					{Region "WA MANAGER LASTRA DA PICKPOINT"}
					(* Ciclo lastra PRELIEVO lastra da punto di prelievo classico *)	
					WAMANAGER_CICLO_PRELIEVO_LASTRA_PP_RUN:
						(* Controllo che la pinza si libera *)
						IF PinzaConProdottoInPresa AND PinzaInQuotaFuoriIngombro THEN
							CmdExe.RapidStopRequest := 1;
							TFError(ErrPRESENZA_MATERIALE_SUPINZA_CICLO_PRELPACCO,ErrNULL,ADR(CmdExe),ADR(State),ADR(Error),ADR(ErrorLog));
						ELSE					
							Mission^.State :=  MISSION_STATE_PRELIEVO_LASTRA_PP_RUN;
						END_IF
							 
					WAMANAGER_CICLO_PRELIEVO_LASTRA_PP_END:;
						 
					(* Ciclo lastra deposito su rulliera *)
					WAMANAGER_CICLO_DEPOSITO_LASTRA_PP_RUN:
						(* Se ho presenza logica *)
						IF ProductOnGripper = KPRODUCTLOADED THEN
							(* Se è abilitato il controllo della presenza utilizzando la fotocellula *)
							IF AbilitaControlloPHGripPresence THEN
								(* Se NON vedo la fotocellula *)
								IF NOT PinzaConProdottoInPresa AND PinzaInQuotaFuoriIngombro THEN
									TFError(ErrLOADLOST,ErrNULL,ADR(CmdExe),ADR(State),ADR(Error),ADR(ErrorLog));
									CmdExe.RapidStopRequest := 1;
									CmdExe.PhaseStopRequest := 1;
								END_IF
							END_IF
						END_IF		
							
						(* Controllo la presenza del pallet nella Postazione di deposito *)	
						IF (Mission^.TPick = TPICK_LASTRA AND NOT IN.PX_WorkArea[Mission^.PPlace]) AND NOT SimulazioneSenzaPalletFalde THEN
							CmdExe.PhaseStopRequest := 1;
							TFError(ErrPALLETNOTPRESENT,Mission^.PPlace,ADR(CmdExe),ADR(State),ADR(Error),ADR(ErrorLog));
						(* Se non ho alcun errore procedo con la missione *)
						ELSIF CmdExe.RapidStopRequest = 0 THEN
							Mission^.State := MISSION_STATE_DEPOSITO_LASTRA_PP_RUN;
						END_IF	
						 
					WAMANAGER_CICLO_DEPOSITO_LASTRA_PP_END:
						 ProductOnGripper := KNOPRODUCT;
				
					{endregion}

					{Region "WA MANAGER LASTRA WA PAL"}		
					WAMANAGER_CICLO_PRELIEVO_LASTRA_WA_RUN:
						(* Controllo che la pinza si libera *)
						IF ((PX_GripPresenceFiltrata AND NOT PX_GripPresenceOK AND AbilitaControlloPHGripPresence) (*OR ProductOnGripper <> KNOPRODUCT*)) AND PinzaInQuotaFuoriIngombro THEN
							CmdExe.RapidStopRequest := 1;
							TFError(ErrPRESENZA_MATERIALE_SUPINZA_CICLO_PRELPACCO,ErrNULL,ADR(CmdExe),ADR(State),ADR(Error),ADR(ErrorLog));
						ELSE					
							Mission^.State :=  MISSION_STATE_PRELIEVO_LASTRA_WA_RUN;	
							PX_GripPresenceOK := TRUE;		
						END_IF					
					WAMANAGER_CICLO_PRELIEVO_LASTRA_WA_END:
						PX_GripPresenceOK := FALSE;
						ProductOnGripper := KPRODUCTLOADED;												
						
					WAMANAGER_CICLO_DEPOSITO_LASTRA_WA_RUN:
						(* Se ho presenza logica *)
						IF ProductOnGripper = KPRODUCTLOADED THEN
							(* Se è abilitato il controllo della presenza utilizzando la fotocellula *)
							IF AbilitaControlloPHGripPresence THEN
								(* Se NON vedo la fotocellula *)
								IF NOT PX_GripPresenceFiltrata AND PinzaInQuotaFuoriIngombro THEN
									TFError(ErrLOADLOST,ErrNULL,ADR(CmdExe),ADR(State),ADR(Error),ADR(ErrorLog));
									CmdExe.RapidStopRequest := 1;
									CmdExe.PhaseStopRequest := 1;
								END_IF
							END_IF
						END_IF		
							
						(* Controllo la presenza del pallet nella Postazione di deposito *)	
						IF (Mission^.TPick = TPICK_PACK AND NOT IN.PX_WorkArea[Mission^.PPlace]) AND NOT SimulazioneSenzaPalletFalde THEN
							CmdExe.PhaseStopRequest := 1;
							TFError(ErrPALLETNOTPRESENT,Mission^.PPlace,ADR(CmdExe),ADR(State),ADR(Error),ADR(ErrorLog));
						(* Se non ho alcun errore procedo con la missione *)
						ELSIF CmdExe.RapidStopRequest = 0 THEN
							Mission^.State := MISSION_STATE_DEPOSITO_LASTRA_WA_RUN;
						END_IF	
						
					WAMANAGER_CICLO_DEPOSITO_LASTRA_WA_END:
						ProductOnGripper := KNOPRODUCT;
					{endregion}	
{region "DEPALLETTIZZATORE"}	
					(* Ciclo lastra PRELIEVO lastra depallettizzatore *)	
					WAMANAGER_CICLO_PRELIEVO_LASTRA_DEPAL_RUN:
						(* Controllo che la pinza si libera *)
						IF ((PX_GripPresenceFiltrata AND NOT PX_GripPresenceOK AND AbilitaControlloPHGripPresence) OR ProductOnGripper <> KNOPRODUCT) AND PinzaInQuotaFuoriIngombro THEN
							CmdExe.RapidStopRequest := 1;
							TFError(ErrPRESENZA_MATERIALE_SUPINZA_CICLO_PRELPACCO,ErrNULL,ADR(CmdExe),ADR(State),ADR(Error),ADR(ErrorLog));
						ELSE					
							Mission^.State :=  MISSION_STATE_PRELIEVO_LASTRA_DEPAL_RUN;	
							PX_GripPresenceOK := TRUE;		
						END_IF
							 
					WAMANAGER_CICLO_PRELIEVO_LASTRA_DEPAL_END:;
						 
					(* Ciclo lastra deposito su rulliera *)
					WAMANAGER_CICLO_DEPOSITO_LASTRA_DEPAL_RUN:
						(* Se ho presenza logica *)
						IF ProductOnGripper = KPRODUCTLOADED THEN
							(* Se è abilitato il controllo della presenza utilizzando la fotocellula *)
							IF AbilitaControlloPHGripPresence THEN
								(* Se NON vedo la fotocellula *)
								IF NOT PX_GripPresenceFiltrata AND PinzaInQuotaFuoriIngombro THEN
									TFError(ErrLOADLOST,ErrNULL,ADR(CmdExe),ADR(State),ADR(Error),ADR(ErrorLog));
									CmdExe.RapidStopRequest := 1;
									CmdExe.PhaseStopRequest := 1;
								END_IF
							END_IF
						END_IF		
							
						(* Controllo la presenza del pallet nella Postazione di deposito *)	
						IF (Mission^.TPick = TPICK_PACK AND NOT IN.PX_WorkArea[Mission^.PPlace]) AND NOT SimulazioneSenzaPalletFalde THEN
							CmdExe.PhaseStopRequest := 1;
							TFError(ErrPALLETNOTPRESENT,Mission^.PPlace,ADR(CmdExe),ADR(State),ADR(Error),ADR(ErrorLog));
						(* Se non ho alcun errore procedo con la missione *)
						ELSIF CmdExe.RapidStopRequest = 0 THEN
							Mission^.State := MISSION_STATE_DEPOSITO_LASTRA_DEPAL_RUN;
						END_IF	
						 
					WAMANAGER_CICLO_DEPOSITO_LASTRA_DEPAL_END:
						 ProductOnGripper := KNOPRODUCT;
							  
					(* Ciclo deposito FALDA su magazzino dedicato dopo prelievo misto da postazione *)
					WAMANAGER_CICLO_DEPOSITO_FALDA_DEPAL_RUN:
						 	
						(* Se ho presenza logica *)
						(*IF ProductOnGripper = KPRODUCTLOADED THEN
							(* Se è abilitato il controllo della presenza utilizzando la fotocellula *)
							IF AbilitaControlloPHGripPresence THEN
								(* Se NON vedo la fotocellula *)
								IF NOT PX_GripPresenceFiltrata AND PinzaInQuotaFuoriIngombro THEN
									TFError(ErrLOADLOST,ErrNULL,ADR(CmdExe),ADR(State),ADR(Error),ADR(ErrorLog));
									CmdExe.RapidStopRequest := 1;
									CmdExe.PhaseStopRequest := 1;
								END_IF
							END_IF
						END_IF*)
							
						IF CmdExe.RapidStopRequest = 0 THEN
							Mission^.State := MISSION_STATE_DEPOSITO_FALDA_DEPAL_RUN;
						END_IF		 
														 
					WAMANAGER_CICLO_DEPOSITO_FALDA_DEPAL_END:
						ProductOnGripper := KNOPRODUCT;	
{endregion}													
				END_CASE
				
{region "CASE MISSION"}		
				(* Eseguo il passo della Missione *)
				CASE Mission^.State OF					
					MISSION_STATE_NOP:
						(* Missione di NOP - WorkFlow  *)
						IF MissionStateCase^.Mission <> MISSION_STATE_NOP THEN
							MissionStateCase^.NCase := 0;
							MissionStateCase^.Mission := MISSION_STATE_NOP;
						END_IF
						
						CASE MissionStateCase^.NCase OF
							(* Case 0 - *)
							0:	
								MissionStateCase^.NCase := 0;
						END_CASE
												
					MISSION_STATE_INIT:
						(* Missione di INIT - WorkFlow  *)
						IF MissionStateCase^.Mission <> MISSION_STATE_INIT THEN
							MissionStateCase^.NCase := 0;
							MissionStateCase^.Mission := MISSION_STATE_INIT;
						END_IF
				{Region "MISSION RIPOSO"}						
					MISSION_STATE_VAIaRIPOSO_RUN:// Assegnato al WorkFlow 2
						(* Missione di RIPOSO - WorkFlow  *)
						NumeroWF := 2;//Numero del WorkFlow
						IF ((MissionStateCase^.Mission <> MISSION_STATE_VAIaRIPOSO_RUN AND MissionStateCase^.Mission <> MISSION_STATE_VAIaRIPOSO_END) AND NOT ForzaPrelievoPaccoDuranteCicloDiRiposo)  THEN
							MissionStateCase^.NCase := 0;
							MissionStateCase^.Mission := MISSION_STATE_VAIaRIPOSO_RUN;
						ELSIF ForzaPrelievoPaccoDuranteCicloDiRiposo THEN
							WorkFlow[NumeroWF].Enable := FALSE;
							MissionStateCase^.NCase := 10;
							Ciclo_Di_Riposo.Stato := INTERROTTO;
						END_IF	
												
						CASE MissionStateCase^.NCase OF
							(* Case 0 - Attivazione e inizializzazione del Workflow*)
							0:	WorkFlow[NumeroWF].Enable := TRUE;
								TFWorkFlowCase(ADR(WorkFlow[NumeroWF]),0,WorkflowCase_JMP);
								MissionStateCase^.NCase := 1;
				
							(* Case 1 - Attesa di un eventuale stop rapido/stop in fase o attesa del completamento/errore workflow *)
							1:	IF CmdExe.RapidStopRequest > 0 OR
									(NOT WorkFlow[NumeroWF].Enable OR WorkFlow[NumeroWF].WFCase = StateWF_ERROR) THEN
									MissionStateCase^.NCase := 2;
								END_IF;
				
							(* Case 2 - Wait WF End *)
							2: IF (NOT WorkFlow[NumeroWF].Enable OR WorkFlow[NumeroWF].State = StateWF_END OR WorkFlow[NumeroWF].WFCase = StateWF_ERROR) THEN
									WorkFlow[NumeroWF].Enable := FALSE;
									IF WorkFlow[NumeroWF].WFCase = StateWF_ERROR THEN
										IF Warning.Code <> ErrNULL THEN
											TFError(Warning.Code,ErrNULL,ADR(CmdExe),ADR(State),ADR(Error),ADR(ErrorLog));
										ELSE
											TFError(ErrWF,ErrNULL,ADR(CmdExe),ADR(State),ADR(Error),ADR(ErrorLog));
										END_IF
									ELSIF WorkFlow[NumeroWF].State = StateWF_END THEN
										MissionStateCase^.NCase := 10;
									ELSE
										(*Invio comando di stop ai moduli*)
										TFParametersArrayClear(ADR (ParametersArray));
										TFPalletizerModulesCommandSend(CmdSTOP,ParametersArray,Modules);
										MissionStateCase^.NCase := 0;
										IF TFIsModuleWarning(Warning) THEN
											TFError(Warning.Code,ErrNULL,ADR(CmdExe),ADR(State),ADR(Error),ADR(ErrorLog));
										END_IF
									END_IF
								END_IF	
							
							(* Case finale *)
							10:
								Mission^.State := MISSION_STATE_VAIaRIPOSO_END;
						END_CASE							 
					MISSION_STATE_VAIaRIPOSO_END:
						(* Missione di RIPOSO TERMINATA - WorkFlow  *)
						IF MissionStateCase^.Mission <> MISSION_STATE_VAIaRIPOSO_END THEN
							MissionStateCase^.NCase := 0;
							MissionStateCase^.Mission := MISSION_STATE_VAIaRIPOSO_END;
						END_IF	
				{ENDREGION}																		
				{Region "MISSION FALDA"}
					MISSION_STATE_PRELIEVO_FALDA_RUN:// Assegnato al WorkFlow 3
						(* Missione di prelievo falda- WorkFlow  *)
						NumeroWF := 3;//Numero del WorkFlow
						IF MissionStateCase^.Mission <> MISSION_STATE_PRELIEVO_FALDA_RUN  AND MissionStateCase^.Mission <> MISSION_STATE_PRELIEVO_FALDA_END THEN
							MissionStateCase^.NCase := 0;
							MissionStateCase^.Mission := MISSION_STATE_PRELIEVO_FALDA_RUN;
						END_IF
																
						CASE MissionStateCase^.NCase OF
							(* Case 0 - Attivazione e inizializzazione del Workflow*)
							0:	WorkFlow[NumeroWF].Enable := TRUE;
								TFWorkFlowCase(ADR(WorkFlow[NumeroWF]),0,WorkflowCase_JMP);
								MissionStateCase^.NCase := 1;
				
							(* Case 1 - Attesa di un eventuale stop rapido/stop in fase o attesa del completamento/errore workflow *)
							1:	IF CmdExe.RapidStopRequest > 0 OR
									(NOT WorkFlow[NumeroWF].Enable OR WorkFlow[NumeroWF].WFCase = StateWF_ERROR) THEN
									MissionStateCase^.NCase := 2;
								END_IF;
				
							(* Case 2 - Wait WF End *)
							2: IF (NOT WorkFlow[NumeroWF].Enable OR WorkFlow[NumeroWF].State = StateWF_END OR WorkFlow[NumeroWF].WFCase = StateWF_ERROR) THEN
								WorkFlow[NumeroWF].Enable := FALSE;
								IF WorkFlow[NumeroWF].WFCase = StateWF_ERROR THEN
									IF Warning.Code <> ErrNULL THEN
										TFError(Warning.Code,ErrNULL,ADR(CmdExe),ADR(State),ADR(Error),ADR(ErrorLog));
									ELSE
										TFError(ErrWF,ErrNULL,ADR(CmdExe),ADR(State),ADR(Error),ADR(ErrorLog));
									END_IF
								ELSIF WorkFlow[NumeroWF].State = StateWF_END THEN
									MissionStateCase^.NCase := 10;
								ELSE
									(*Invio comando di stop ai moduli*)
									TFParametersArrayClear(ADR (ParametersArray));
									TFPalletizerModulesCommandSend(CmdSTOP,ParametersArray,Modules);
									MissionStateCase^.NCase := 0;
									IF TFIsModuleWarning(Warning) THEN
										TFError(Warning.Code,ErrNULL,ADR(CmdExe),ADR(State),ADR(Error),ADR(ErrorLog));
									END_IF
								END_IF
							END_IF
							
							(* Case finale *)
							10:	
								Mission^.State := MISSION_STATE_PRELIEVO_FALDA_END;
								
						END_CASE
						
					MISSION_STATE_PRELIEVO_FALDA_END:
						(* Missione TERMINATA - WorkFlow  *)
						IF MissionStateCase^.Mission <> MISSION_STATE_PRELIEVO_FALDA_END THEN
							MissionStateCase^.NCase := 0;
							MissionStateCase^.Mission := MISSION_STATE_PRELIEVO_FALDA_END;
						END_IF
						
						CASE MissionStateCase^.NCase OF
							(* Case 0 - *)
							0:  Mission^.State := MISSION_STATE_PRELIEVO_FALDA_END;
								MissionStateCase^.NCase := 0;
						END_CASE	
					
					MISSION_STATE_DEPOSITO_FALDA_RUN: // Assegnato al WorkFlow 4
						NumeroWF:=4;//Numero del WorkFlow
						IF MissionStateCase^.Mission <> MISSION_STATE_DEPOSITO_FALDA_RUN  AND MissionStateCase^.Mission <> MISSION_STATE_DEPOSITO_FALDA_END THEN
							MissionStateCase^.NCase := 0;
							MissionStateCase^.Mission := MISSION_STATE_DEPOSITO_FALDA_RUN;
						END_IF
						
						CASE MissionStateCase^.NCase OF
						(* Case 0 - Attivazione e inizializzazione del Workflow*)
							0:	WorkFlow[NumeroWF].Enable := TRUE;
								TFWorkFlowCase(ADR(WorkFlow[NumeroWF]),0,WorkflowCase_JMP);
								MissionStateCase^.NCase := 1;
				
							(* Case 1 - Attesa di un eventuale stop rapido/stop in fase o attesa del completamento/errore workflow *)
							1:	IF CmdExe.RapidStopRequest > 0 OR
									(NOT WorkFlow[NumeroWF].Enable OR WorkFlow[NumeroWF].WFCase = StateWF_ERROR) THEN
									MissionStateCase^.NCase := 2;
								END_IF;
				
							(* Case 2 - Wait WF End *)
							2: IF (NOT WorkFlow[NumeroWF].Enable OR WorkFlow[NumeroWF].State = StateWF_END OR WorkFlow[NumeroWF].WFCase = StateWF_ERROR) THEN
									WorkFlow[NumeroWF].Enable := FALSE;
									IF WorkFlow[NumeroWF].WFCase = StateWF_ERROR THEN
										IF Warning.Code <> ErrNULL THEN
											TFError(Warning.Code,ErrNULL,ADR(CmdExe),ADR(State),ADR(Error),ADR(ErrorLog));
										ELSE
											TFError(ErrWF,ErrNULL,ADR(CmdExe),ADR(State),ADR(Error),ADR(ErrorLog));
										END_IF
									ELSIF WorkFlow[NumeroWF].State = StateWF_END THEN
										MissionStateCase^.NCase := 10;
									ELSE
										(*Invio comando di stop ai moduli*)
										TFParametersArrayClear(ADR (ParametersArray));
										TFPalletizerModulesCommandSend(CmdSTOP,ParametersArray,Modules);
										MissionStateCase^.NCase := 0;
										IF TFIsModuleWarning(Warning) THEN
											TFError(Warning.Code,ErrNULL,ADR(CmdExe),ADR(State),ADR(Error),ADR(ErrorLog));
										END_IF
									END_IF
								END_IF
								
							(* Case finale *)
							10:
								Mission^.State := MISSION_STATE_DEPOSITO_FALDA_END;
								
						END_CASE
						
					MISSION_STATE_DEPOSITO_FALDA_END:					
						IF MissionStateCase^.Mission <> MISSION_STATE_DEPOSITO_FALDA_END THEN
							MissionStateCase^.NCase := 0;
							MissionStateCase^.Mission := MISSION_STATE_DEPOSITO_FALDA_END;
						END_IF
						
						CASE MissionStateCase^.NCase OF
							(* Case 0 - *)
							0:  Mission^.State := MISSION_STATE_DEPOSITO_FALDA_END;
								MissionStateCase^.NCase := 0;
						END_CASE	
				{ENDREGION}																		
				{Region "MISSION LASTRA DA PICKPOINT"}
				MISSION_STATE_PRELIEVO_LASTRA_PP_RUN:
						NumeroWF:= 5  ;//Numero del WorkFlow				
						IF MissionStateCase^.Mission <> MISSION_STATE_PRELIEVO_LASTRA_PP_RUN  AND MissionStateCase^.Mission <> MISSION_STATE_PRELIEVO_LASTRA_PP_END THEN
							MissionStateCase^.NCase := 0;
							MissionStateCase^.Mission := MISSION_STATE_PRELIEVO_LASTRA_PP_RUN;
						END_IF
						
						CASE MissionStateCase^.NCase OF
							(* Case 0 - Attivazione e inizializzazione del Workflow*)
							0:	WorkFlow[NumeroWF].Enable := TRUE;
								TFWorkFlowCase(ADR(WorkFlow[NumeroWF]),0,WorkflowCase_JMP);
								MissionStateCase^.NCase := 1;
				
							(* Case 1 - Attesa di un eventuale stop rapido/stop in fase o attesa del completamento/errore workflow *)
							1:	IF CmdExe.RapidStopRequest > 0 OR
									(NOT WorkFlow[NumeroWF].Enable OR WorkFlow[NumeroWF].WFCase = StateWF_ERROR) THEN
									MissionStateCase^.NCase := 2;
								END_IF;
				
							(* Case 2 - Wait WF End *)
							2: IF (NOT WorkFlow[NumeroWF].Enable OR WorkFlow[NumeroWF].State = StateWF_END OR WorkFlow[NumeroWF].WFCase = StateWF_ERROR) THEN
									WorkFlow[NumeroWF].Enable := FALSE;
									IF WorkFlow[NumeroWF].WFCase = StateWF_ERROR THEN
										IF Warning.Code <> ErrNULL THEN
											TFError(Warning.Code,ErrNULL,ADR(CmdExe),ADR(State),ADR(Error),ADR(ErrorLog));
										ELSE
											TFError(ErrWF,ErrNULL,ADR(CmdExe),ADR(State),ADR(Error),ADR(ErrorLog));
										END_IF
									ELSIF WorkFlow[NumeroWF].State = StateWF_END THEN
										MissionStateCase^.NCase := 10;
									ELSE
										(*Invio comando di stop ai moduli*)
										TFParametersArrayClear(ADR (ParametersArray));
										TFPalletizerModulesCommandSend(CmdSTOP,ParametersArray,Modules);
										MissionStateCase^.NCase := 0;
										IF TFIsModuleWarning(Warning) THEN
											TFError(Warning.Code,ErrNULL,ADR(CmdExe),ADR(State),ADR(Error),ADR(ErrorLog));
										END_IF
									END_IF
								END_IF
								
							(* Case finale *)
							10:
								Mission^.State := MISSION_STATE_PRELIEVO_LASTRA_PP_END;
									
						END_CASE				
					MISSION_STATE_PRELIEVO_LASTRA_PP_END:
						IF MissionStateCase^.Mission <> MISSION_STATE_PRELIEVO_LASTRA_PP_END THEN
							MissionStateCase^.NCase := 0;
							MissionStateCase^.Mission := MISSION_STATE_PRELIEVO_LASTRA_PP_END;
						END_IF
						
						CASE MissionStateCase^.NCase OF
							
							(* Case 0 - *)
							0:  Mission^.State := MISSION_STATE_PRELIEVO_LASTRA_PP_END;
							
						END_CASE					
					MISSION_STATE_DEPOSITO_LASTRA_PP_RUN:
						NumeroWF:= 6;//Numero del WorkFlow				
						IF MissionStateCase^.Mission <> MISSION_STATE_DEPOSITO_LASTRA_PP_RUN  AND MissionStateCase^.Mission <> MISSION_STATE_DEPOSITO_LASTRA_PP_RUN THEN
							MissionStateCase^.NCase := 0;
							MissionStateCase^.Mission := MISSION_STATE_DEPOSITO_LASTRA_PP_RUN;
						END_IF
						
						CASE MissionStateCase^.NCase OF
							(* Case 0 - Attivazione e inizializzazione del Workflow*)
							0:	WorkFlow[NumeroWF].Enable := TRUE;
								TFWorkFlowCase(ADR(WorkFlow[NumeroWF]),0,WorkflowCase_JMP);
								MissionStateCase^.NCase := 1;
				
							(* Case 1 - Attesa di un eventuale stop rapido/stop in fase o attesa del completamento/errore workflow *)
							1:	IF CmdExe.RapidStopRequest > 0 OR
									(NOT WorkFlow[NumeroWF].Enable OR WorkFlow[NumeroWF].WFCase = StateWF_ERROR) THEN
									MissionStateCase^.NCase := 2;
								END_IF;
				
							(* Case 2 - Wait WF End *)
							2: IF (NOT WorkFlow[NumeroWF].Enable OR WorkFlow[NumeroWF].State = StateWF_END OR WorkFlow[NumeroWF].WFCase = StateWF_ERROR) THEN
									//IF (Ciclo_Deposito_Lastra_Depal.Passo = 56 AND Ciclo_Deposito_Lastra_Depal.Stato = INTERROTTO) OR StopDepositoPerArresto THEN
									//	WorkFlow[NumeroWF].Enable := TRUE;
									//ELSE
										WorkFlow[NumeroWF].Enable := FALSE;
									//END_IF
									IF WorkFlow[NumeroWF].WFCase = StateWF_ERROR THEN
										IF Warning.Code <> ErrNULL THEN
											TFError(Warning.Code,ErrNULL,ADR(CmdExe),ADR(State),ADR(Error),ADR(ErrorLog));
										ELSE
											TFError(ErrWF,ErrNULL,ADR(CmdExe),ADR(State),ADR(Error),ADR(ErrorLog));
										END_IF
									ELSIF WorkFlow[NumeroWF].State = StateWF_END THEN//AND NOT StopDepositoPerArresto THEN
										MissionStateCase^.NCase := 10;
									ELSE
										(*Invio comando di stop ai moduli*)
										TFParametersArrayClear(ADR (ParametersArray));
										TFPalletizerModulesCommandSend(CmdSTOP,ParametersArray,Modules);
										IF TFIsModuleWarning(Warning) THEN
											TFError(Warning.Code,ErrNULL,ADR(CmdExe),ADR(State),ADR(Error),ADR(ErrorLog));
										END_IF
									END_IF
								END_IF
								
							(* Case finale *)
							10:
								Mission^.State := MISSION_STATE_DEPOSITO_LASTRA_PP_END;
									
						END_CASE					
					MISSION_STATE_DEPOSITO_LASTRA_PP_END:
						IF MissionStateCase^.Mission <> MISSION_STATE_DEPOSITO_LASTRA_PP_END THEN
							MissionStateCase^.NCase := 0;
							MissionStateCase^.Mission := MISSION_STATE_DEPOSITO_LASTRA_PP_END;
						END_IF
						
						CASE MissionStateCase^.NCase OF
							
							(* Case 0 - *)
							0:  Mission^.State := MISSION_STATE_DEPOSITO_LASTRA_PP_END;
							
						END_CASE

				{endregion}

				{Region "MISSION LASTRA WA"}
					MISSION_STATE_PRELIEVO_LASTRA_WA_RUN:// Assegnato al WorkFlow 7
						NumeroWF:=7;//Numero del WorkFlow
						IF MissionStateCase^.Mission <> MISSION_STATE_PRELIEVO_LASTRA_WA_RUN AND MissionStateCase^.Mission <> MISSION_STATE_PRELIEVO_LASTRA_WA_END THEN
							MissionStateCase^.NCase := 0;
							MissionStateCase^.Mission := MISSION_STATE_PRELIEVO_LASTRA_WA_RUN;
						END_IF
	 					//
						CASE MissionStateCase^.NCase OF
							(* Case 0 - Attivazione e inizializzazione del Workflow*)
							0:	WorkFlow[NumeroWF].Enable := TRUE;
								TFWorkFlowCase(ADR(WorkFlow[NumeroWF]),0,WorkflowCase_JMP);
								MissionStateCase^.NCase := 1;			
							(* Case 1 - Attesa di un eventuale stop rapido/stop in fase o attesa del completamento/errore workflow *)
							1:	IF CmdExe.RapidStopRequest > 0 OR
									(NOT WorkFlow[NumeroWF].Enable OR WorkFlow[NumeroWF].WFCase = StateWF_ERROR) THEN
									MissionStateCase^.NCase := 2;
								END_IF;			
							(* Case 2 - Wait WF End *)
							2: IF (NOT WorkFlow[NumeroWF].Enable OR WorkFlow[NumeroWF].State = StateWF_END OR WorkFlow[NumeroWF].WFCase = StateWF_ERROR) THEN
									WorkFlow[NumeroWF].Enable := FALSE;
									IF WorkFlow[NumeroWF].WFCase = StateWF_ERROR THEN
										IF Warning.Code <> ErrNULL THEN
											TFError(Warning.Code,ErrNULL,ADR(CmdExe),ADR(State),ADR(Error),ADR(ErrorLog));
										ELSE
											TFError(ErrWF,ErrNULL,ADR(CmdExe),ADR(State),ADR(Error),ADR(ErrorLog));
										END_IF
									ELSIF WorkFlow[NumeroWF].State = StateWF_END THEN
										MissionStateCase^.NCase := 10;
									ELSE
										(*Invio comando di stop ai moduli*)
										TFParametersArrayClear(ADR (ParametersArray));
										TFPalletizerModulesCommandSend(CmdSTOP,ParametersArray,Modules);
										MissionStateCase^.NCase := 0;
										IF TFIsModuleWarning(Warning) THEN
											TFError(Warning.Code,ErrNULL,ADR(CmdExe),ADR(State),ADR(Error),ADR(ErrorLog));
										END_IF
									END_IF
								END_IF
								
							(* Case finale *)
							10:
								Mission^.State := MISSION_STATE_PRELIEVO_LASTRA_WA_END;							
						END_CASE
						
					MISSION_STATE_PRELIEVO_LASTRA_WA_END:
						IF MissionStateCase^.Mission <> MISSION_STATE_PRELIEVO_LASTRA_WA_END THEN
							MissionStateCase^.NCase := 0;
							MissionStateCase^.Mission := MISSION_STATE_PRELIEVO_LASTRA_WA_END;
						END_IF
						
						CASE MissionStateCase^.NCase OF
							
							(* Case 0 - *)
							0:  Mission^.State := MISSION_STATE_PRELIEVO_LASTRA_WA_END;
								MissionStateCase^.NCase := 0;
													
						END_CASE		
				{ENDREGION}																		
				{Region "MISSION LASTRA PAREGGIATORE"}
					MISSION_STATE_DEPOSITO_LASTRA_SU_PAREGGIATORE_RUN:// Assegnato al WorkFlow 6
						NumeroWF:=8;//Numero del WorkFlow
						IF MissionStateCase^.Mission <> MISSION_STATE_DEPOSITO_LASTRA_SU_PAREGGIATORE_RUN AND MissionStateCase^.Mission <> MISSION_STATE_DEPOSITO_LASTRA_SU_PAREGGIATORE_END THEN
							MissionStateCase^.NCase := 0;
							MissionStateCase^.Mission := MISSION_STATE_DEPOSITO_LASTRA_SU_PAREGGIATORE_RUN;
						END_IF
						CASE MissionStateCase^.NCase OF
							(* Case 0 - Attivazione e inizializzazione del Workflow*)
							0:	WorkFlow[NumeroWF].Enable := TRUE;
								TFWorkFlowCase(ADR(WorkFlow[NumeroWF]),0,WorkflowCase_JMP);
								MissionStateCase^.NCase := 1;
							(* Case 1 - Attesa di un eventuale stop rapido/stop in fase o attesa del completamento/errore workflow *)
							1:	IF CmdExe.RapidStopRequest > 0 OR
									(NOT WorkFlow[NumeroWF].Enable OR WorkFlow[NumeroWF].WFCase = StateWF_ERROR) THEN
									MissionStateCase^.NCase := 2;
								END_IF;
							(* Case 2 - Wait WF End *)
							2: IF (NOT WorkFlow[NumeroWF].Enable OR WorkFlow[NumeroWF].State = StateWF_END OR WorkFlow[NumeroWF].WFCase = StateWF_ERROR) THEN
									WorkFlow[NumeroWF].Enable := FALSE;
									IF WorkFlow[NumeroWF].WFCase = StateWF_ERROR THEN
										IF Warning.Code <> ErrNULL THEN
											TFError(Warning.Code,ErrNULL,ADR(CmdExe),ADR(State),ADR(Error),ADR(ErrorLog));
										ELSE
											TFError(ErrWF,ErrNULL,ADR(CmdExe),ADR(State),ADR(Error),ADR(ErrorLog));
										END_IF
									ELSIF WorkFlow[NumeroWF].State = StateWF_END THEN
										MissionStateCase^.NCase := 10;
									ELSE
										(*Invio comando di stop ai moduli*)
										TFParametersArrayClear(ADR (ParametersArray));
										TFPalletizerModulesCommandSend(CmdSTOP,ParametersArray,Modules);
										MissionStateCase^.NCase := 0;
										IF TFIsModuleWarning(Warning) THEN
											TFError(Warning.Code,ErrNULL,ADR(CmdExe),ADR(State),ADR(Error),ADR(ErrorLog));
										END_IF
									END_IF
								END_IF
							(* Case finale *)
							10:
								Mission^.State := MISSION_STATE_DEPOSITO_LASTRA_SU_PAREGGIATORE_END;
						END_CASE
							 
					MISSION_STATE_DEPOSITO_LASTRA_SU_PAREGGIATORE_END:
						IF MissionStateCase^.Mission <> MISSION_STATE_DEPOSITO_LASTRA_SU_PAREGGIATORE_END THEN
							MissionStateCase^.NCase := 0;
							MissionStateCase^.Mission := MISSION_STATE_DEPOSITO_LASTRA_SU_PAREGGIATORE_END;
						END_IF
						
						CASE MissionStateCase^.NCase OF
							(* Case 0 - *)
							0:  Mission^.State := MISSION_STATE_DEPOSITO_LASTRA_SU_PAREGGIATORE_END;
								MissionStateCase^.NCase := 0;
						END_CASE
						
					MISSION_STATE_PRELIEVO_LASTRA_DA_PAREGGIATORE_RUN:// Assegnato al WorkFlow 7
						NumeroWF:=7;//Numero del WorkFlow
						IF MissionStateCase^.Mission <> MISSION_STATE_PRELIEVO_LASTRA_DA_PAREGGIATORE_RUN AND MissionStateCase^.Mission <> MISSION_STATE_PRELIEVO_LASTRA_DA_PAREGGIATORE_END THEN
							MissionStateCase^.NCase := 0;
							MissionStateCase^.Mission := MISSION_STATE_PRELIEVO_LASTRA_WA_RUN;
						END_IF			
						CASE MissionStateCase^.NCase OF
							(* Case 0 - Attivazione e inizializzazione del Workflow*)
							0:	WorkFlow[NumeroWF].Enable := TRUE;
								TFWorkFlowCase(ADR(WorkFlow[NumeroWF]),0,WorkflowCase_JMP);
								MissionStateCase^.NCase := 1;
							(* Case 1 - Attesa di un eventuale stop rapido/stop in fase o attesa del completamento/errore workflow *)
							1:	IF CmdExe.RapidStopRequest > 0 OR
									(NOT WorkFlow[NumeroWF].Enable OR WorkFlow[NumeroWF].WFCase = StateWF_ERROR) THEN
									MissionStateCase^.NCase := 2;
								END_IF;
							(* Case 2 - Wait WF End *)
							2: IF (NOT WorkFlow[NumeroWF].Enable OR WorkFlow[NumeroWF].State = StateWF_END OR WorkFlow[NumeroWF].WFCase = StateWF_ERROR) THEN
									WorkFlow[NumeroWF].Enable := FALSE;
									IF WorkFlow[NumeroWF].WFCase = StateWF_ERROR THEN
										IF Warning.Code <> ErrNULL THEN
											TFError(Warning.Code,ErrNULL,ADR(CmdExe),ADR(State),ADR(Error),ADR(ErrorLog));
										ELSE
											TFError(ErrWF,ErrNULL,ADR(CmdExe),ADR(State),ADR(Error),ADR(ErrorLog));
										END_IF
									ELSIF WorkFlow[NumeroWF].State = StateWF_END THEN
										MissionStateCase^.NCase := 10;
									ELSE
										(*Invio comando di stop ai moduli*)
										TFParametersArrayClear(ADR (ParametersArray));
										TFPalletizerModulesCommandSend(CmdSTOP,ParametersArray,Modules);
										MissionStateCase^.NCase := 0;
										IF TFIsModuleWarning(Warning) THEN
											TFError(Warning.Code,ErrNULL,ADR(CmdExe),ADR(State),ADR(Error),ADR(ErrorLog));
										END_IF
									END_IF
								END_IF
							(* Case finale *)
							10:
								Mission^.State := MISSION_STATE_PRELIEVO_LASTRA_WA_END;
						END_CASE
					MISSION_STATE_PRELIEVO_LASTRA_DA_PAREGGIATORE_END:
						IF MissionStateCase^.Mission <> MISSION_STATE_PRELIEVO_LASTRA_DA_PAREGGIATORE_END THEN
							MissionStateCase^.NCase := 0;
							MissionStateCase^.Mission := MISSION_STATE_PRELIEVO_LASTRA_DA_PAREGGIATORE_END;
						END_IF
						
						CASE MissionStateCase^.NCase OF
							(* Case 0 - *)
							0:  Mission^.State := MISSION_STATE_PRELIEVO_LASTRA_DA_PAREGGIATORE_END;
								MissionStateCase^.NCase := 0;
						END_CASE
				{ENDREGION}																		
				{Region "MISSION DEPOSITO LASTRA WA"}											
					MISSION_STATE_DEPOSITO_LASTRA_WA_RUN:// Assegnato al WorkFlow 
						NumeroWF:=9;//Numero del WorkFlow				
						IF MissionStateCase^.Mission <> MISSION_STATE_DEPOSITO_LASTRA_WA_RUN  AND MissionStateCase^.Mission <> MISSION_STATE_DEPOSITO_LASTRA_WA_END THEN
							MissionStateCase^.NCase := 0;
							MissionStateCase^.Mission := MISSION_STATE_DEPOSITO_LASTRA_WA_RUN;
						END_IF
						CASE MissionStateCase^.NCase OF
							(* Case 0 - Attivazione e inizializzazione del Workflow*)
							0:	WorkFlow[NumeroWF].Enable := TRUE;
								TFWorkFlowCase(ADR(WorkFlow[NumeroWF]),0,WorkflowCase_JMP);
								MissionStateCase^.NCase := 1;
							(* Case 1 - Attesa di un eventuale stop rapido/stop in fase o attesa del completamento/errore workflow *)
							1:	IF CmdExe.RapidStopRequest > 0 OR
									(NOT WorkFlow[NumeroWF].Enable OR WorkFlow[NumeroWF].WFCase = StateWF_ERROR) THEN
									MissionStateCase^.NCase := 2;
								END_IF;
							(* Case 2 - Wait WF End *)
							2: IF (NOT WorkFlow[NumeroWF].Enable OR WorkFlow[NumeroWF].State = StateWF_END OR WorkFlow[NumeroWF].WFCase = StateWF_ERROR) THEN
									WorkFlow[NumeroWF].Enable := FALSE;
									IF WorkFlow[NumeroWF].WFCase = StateWF_ERROR THEN
										IF Warning.Code <> ErrNULL THEN
											TFError(Warning.Code,ErrNULL,ADR(CmdExe),ADR(State),ADR(Error),ADR(ErrorLog));
										ELSE
											TFError(ErrWF,ErrNULL,ADR(CmdExe),ADR(State),ADR(Error),ADR(ErrorLog));
										END_IF
									ELSIF WorkFlow[NumeroWF].State = StateWF_END THEN
										MissionStateCase^.NCase := 10;
									ELSE
										(*Invio comando di stop ai moduli*)
										TFParametersArrayClear(ADR (ParametersArray));
										TFPalletizerModulesCommandSend(CmdSTOP,ParametersArray,Modules);
										MissionStateCase^.NCase := 0;
										IF TFIsModuleWarning(Warning) THEN
											TFError(Warning.Code,ErrNULL,ADR(CmdExe),ADR(State),ADR(Error),ADR(ErrorLog));
										END_IF
									END_IF
								END_IF
							(* Case finale *)
							10:
								Mission^.State := MISSION_STATE_DEPOSITO_LASTRA_WA_END;
						END_CASE
						
					MISSION_STATE_DEPOSITO_LASTRA_WA_END:	
						IF MissionStateCase^.Mission <> MISSION_STATE_DEPOSITO_LASTRA_WA_END THEN
							MissionStateCase^.NCase := 0;
							MissionStateCase^.Mission := MISSION_STATE_DEPOSITO_LASTRA_WA_END;
						END_IF
						
						CASE MissionStateCase^.NCase OF
							
							(* Case 0 - *)
							0:  Mission^.State := MISSION_STATE_DEPOSITO_LASTRA_WA_END;
							
						END_CASE
					{ENDREGION}																		
																		
				{Region "MISSION DEPAL"}			
					MISSION_STATE_PRELIEVO_LASTRA_DEPAL_RUN:
						NumeroWF:=10;//Numero del WorkFlow				
						IF MissionStateCase^.Mission <> MISSION_STATE_PRELIEVO_LASTRA_DEPAL_RUN  AND MissionStateCase^.Mission <> MISSION_STATE_PRELIEVO_LASTRA_DEPAL_END THEN
							MissionStateCase^.NCase := 0;
							MissionStateCase^.Mission := MISSION_STATE_PRELIEVO_LASTRA_DEPAL_RUN;
						END_IF
						
						CASE MissionStateCase^.NCase OF
							(* Case 0 - Attivazione e inizializzazione del Workflow*)
							0:	WorkFlow[NumeroWF].Enable := TRUE;
								TFWorkFlowCase(ADR(WorkFlow[NumeroWF]),0,WorkflowCase_JMP);
								MissionStateCase^.NCase := 1;
				
							(* Case 1 - Attesa di un eventuale stop rapido/stop in fase o attesa del completamento/errore workflow *)
							1:	IF CmdExe.RapidStopRequest > 0 OR
									(NOT WorkFlow[NumeroWF].Enable OR WorkFlow[NumeroWF].WFCase = StateWF_ERROR) THEN
									MissionStateCase^.NCase := 2;
								END_IF;
				
							(* Case 2 - Wait WF End *)
							2: IF (NOT WorkFlow[NumeroWF].Enable OR WorkFlow[NumeroWF].State = StateWF_END OR WorkFlow[NumeroWF].WFCase = StateWF_ERROR) THEN
									WorkFlow[NumeroWF].Enable := FALSE;
									IF WorkFlow[NumeroWF].WFCase = StateWF_ERROR THEN
										IF Warning.Code <> ErrNULL THEN
											TFError(Warning.Code,ErrNULL,ADR(CmdExe),ADR(State),ADR(Error),ADR(ErrorLog));
										ELSE
											TFError(ErrWF,ErrNULL,ADR(CmdExe),ADR(State),ADR(Error),ADR(ErrorLog));
										END_IF
									ELSIF WorkFlow[NumeroWF].State = StateWF_END THEN
										MissionStateCase^.NCase := 10;
									ELSE
										(*Invio comando di stop ai moduli*)
										TFParametersArrayClear(ADR (ParametersArray));
										TFPalletizerModulesCommandSend(CmdSTOP,ParametersArray,Modules);
										MissionStateCase^.NCase := 0;
										IF TFIsModuleWarning(Warning) THEN
											TFError(Warning.Code,ErrNULL,ADR(CmdExe),ADR(State),ADR(Error),ADR(ErrorLog));
										END_IF
									END_IF
								END_IF
								
							(* Case finale *)
							10:
								Mission^.State := MISSION_STATE_PRELIEVO_LASTRA_DEPAL_END;
									
						END_CASE				
					MISSION_STATE_PRELIEVO_LASTRA_DEPAL_END:
						IF MissionStateCase^.Mission <> MISSION_STATE_PRELIEVO_LASTRA_DEPAL_END THEN
							MissionStateCase^.NCase := 0;
							MissionStateCase^.Mission := MISSION_STATE_PRELIEVO_LASTRA_DEPAL_END;
						END_IF
						
						CASE MissionStateCase^.NCase OF
							
							(* Case 0 - *)
							0:  Mission^.State := MISSION_STATE_PRELIEVO_LASTRA_DEPAL_END;
							
						END_CASE					
					MISSION_STATE_DEPOSITO_LASTRA_DEPAL_RUN:
						NumeroWF:=12;//Numero del WorkFlow				
						IF MissionStateCase^.Mission <> MISSION_STATE_DEPOSITO_LASTRA_DEPAL_RUN  AND MissionStateCase^.Mission <> MISSION_STATE_DEPOSITO_LASTRA_DEPAL_END THEN
							MissionStateCase^.NCase := 0;
							MissionStateCase^.Mission := MISSION_STATE_DEPOSITO_LASTRA_DEPAL_RUN;
						END_IF
						
						CASE MissionStateCase^.NCase OF
							(* Case 0 - Attivazione e inizializzazione del Workflow*)
							0:	WorkFlow[NumeroWF].Enable := TRUE;
								TFWorkFlowCase(ADR(WorkFlow[NumeroWF]),0,WorkflowCase_JMP);
								MissionStateCase^.NCase := 1;
				
							(* Case 1 - Attesa di un eventuale stop rapido/stop in fase o attesa del completamento/errore workflow *)
							1:	IF CmdExe.RapidStopRequest > 0 OR
									(NOT WorkFlow[NumeroWF].Enable OR WorkFlow[NumeroWF].WFCase = StateWF_ERROR) THEN
									MissionStateCase^.NCase := 2;
								END_IF;
				
							(* Case 2 - Wait WF End *)
							2: IF (NOT WorkFlow[NumeroWF].Enable OR WorkFlow[NumeroWF].State = StateWF_END OR WorkFlow[NumeroWF].WFCase = StateWF_ERROR) THEN
									IF (Ciclo_Deposito_Lastra_Depal.Passo = 56 AND Ciclo_Deposito_Lastra_Depal.Stato = INTERROTTO) OR StopDepositoPerArresto THEN
										WorkFlow[NumeroWF].Enable := TRUE;
									ELSE
										WorkFlow[NumeroWF].Enable := FALSE;
									END_IF
									IF WorkFlow[NumeroWF].WFCase = StateWF_ERROR THEN
										IF Warning.Code <> ErrNULL THEN
											TFError(Warning.Code,ErrNULL,ADR(CmdExe),ADR(State),ADR(Error),ADR(ErrorLog));
										ELSE
											TFError(ErrWF,ErrNULL,ADR(CmdExe),ADR(State),ADR(Error),ADR(ErrorLog));
										END_IF
									ELSIF WorkFlow[NumeroWF].State = StateWF_END AND NOT StopDepositoPerArresto THEN
										MissionStateCase^.NCase := 10;
									ELSE
										(*Invio comando di stop ai moduli*)
										TFParametersArrayClear(ADR (ParametersArray));
										TFPalletizerModulesCommandSend(CmdSTOP,ParametersArray,Modules);
										IF TFIsModuleWarning(Warning) THEN
											TFError(Warning.Code,ErrNULL,ADR(CmdExe),ADR(State),ADR(Error),ADR(ErrorLog));
										END_IF
									END_IF
								END_IF
								
							(* Case finale *)
							10:
								Mission^.State := MISSION_STATE_DEPOSITO_LASTRA_DEPAL_END;
									
						END_CASE					
					MISSION_STATE_DEPOSITO_LASTRA_DEPAL_END:
						IF MissionStateCase^.Mission <> MISSION_STATE_DEPOSITO_LASTRA_DEPAL_END THEN
							MissionStateCase^.NCase := 0;
							MissionStateCase^.Mission := MISSION_STATE_DEPOSITO_LASTRA_DEPAL_END;
						END_IF
						
						CASE MissionStateCase^.NCase OF
							
							(* Case 0 - *)
							0:  Mission^.State := MISSION_STATE_DEPOSITO_LASTRA_DEPAL_END;
							
						END_CASE
					MISSION_STATE_DEPOSITO_FALDA_DEPAL_RUN:
						NumeroWF:=11;//Numero del WorkFlow				
						IF MissionStateCase^.Mission <> MISSION_STATE_DEPOSITO_FALDA_DEPAL_RUN  AND MissionStateCase^.Mission <> MISSION_STATE_DEPOSITO_FALDA_DEPAL_END THEN
							MissionStateCase^.NCase := 0;
							MissionStateCase^.Mission := MISSION_STATE_DEPOSITO_FALDA_DEPAL_RUN;
						END_IF
						
						CASE MissionStateCase^.NCase OF
							(* Case 0 - Attivazione e inizializzazione del Workflow*)
							0:	WorkFlow[NumeroWF].Enable := TRUE;
								TFWorkFlowCase(ADR(WorkFlow[NumeroWF]),0,WorkflowCase_JMP);
								MissionStateCase^.NCase := 1;
				
							(* Case 1 - Attesa di un eventuale stop rapido/stop in fase o attesa del completamento/errore workflow *)
							1:	IF CmdExe.RapidStopRequest > 0 OR
									(NOT WorkFlow[NumeroWF].Enable OR WorkFlow[NumeroWF].WFCase = StateWF_ERROR) THEN
									MissionStateCase^.NCase := 2;
								END_IF;
				
							(* Case 2 - Wait WF End *)
							2: IF (NOT WorkFlow[NumeroWF].Enable OR WorkFlow[NumeroWF].State = StateWF_END OR WorkFlow[NumeroWF].WFCase = StateWF_ERROR) THEN
									WorkFlow[NumeroWF].Enable := FALSE;
									IF WorkFlow[NumeroWF].WFCase = StateWF_ERROR THEN
										IF Warning.Code <> ErrNULL THEN
											TFError(Warning.Code,ErrNULL,ADR(CmdExe),ADR(State),ADR(Error),ADR(ErrorLog));
										ELSE
											TFError(ErrWF,ErrNULL,ADR(CmdExe),ADR(State),ADR(Error),ADR(ErrorLog));
										END_IF
									ELSIF WorkFlow[NumeroWF].State = StateWF_END THEN
										MissionStateCase^.NCase := 10;
									ELSE
										(*Invio comando di stop ai moduli*)
										TFParametersArrayClear(ADR (ParametersArray));
										TFPalletizerModulesCommandSend(CmdSTOP,ParametersArray,Modules);
										MissionStateCase^.NCase := 0;
										IF TFIsModuleWarning(Warning) THEN
											TFError(Warning.Code,ErrNULL,ADR(CmdExe),ADR(State),ADR(Error),ADR(ErrorLog));
										END_IF
									END_IF
								END_IF
								
							(* Case finale *)
							10:
								Mission^.State := MISSION_STATE_DEPOSITO_FALDA_DEPAL_END;
									
						END_CASE					
					MISSION_STATE_DEPOSITO_FALDA_DEPAL_END:
						IF MissionStateCase^.Mission <> MISSION_STATE_DEPOSITO_FALDA_DEPAL_END THEN
							MissionStateCase^.NCase := 0;
							MissionStateCase^.Mission := MISSION_STATE_DEPOSITO_FALDA_DEPAL_END;
						END_IF
						
						CASE MissionStateCase^.NCase OF
							
							(* Case 0 - *)
							0:  Mission^.State := MISSION_STATE_DEPOSITO_FALDA_DEPAL_END;
							
						END_CASE
				{ENDREGION}													  

					MISSION_STATE_ERROR:
						CmdExe.PhaseStopRequest := 1;
						WorkFlow[1].Enable := FALSE;
						
				ELSE;
				END_CASE
			END_IF
			
		(* Case 100 *)
		(* WorkFlow END *)
		100:WorkFlow[1].State := StateWF_END;
			WorkFlow[1].Enable := FALSE;
			TFWorkFlowCase(ADR(WorkFlow[1]),0,WorkflowCase_JMP);
			
		(* Case 999 *)
		(* WorkFlow ERROR *)
		StateWF_ERROR:
			TFWorkFlowError(ADR(WorkFlow[1]),ADR(WorkFlowErrorLog[1]));
			WorkFlow[1].Enable := FALSE;

		ELSE
			TFWorkFlowError(ADR(WorkFlow[1]),ADR(WorkFlowErrorLog[1]));
			TFError(ErrNOCMDCASE,ErrNULL,ADR(CmdExe),ADR(State),ADR(Error),ADR(ErrorLog));

	END_CASE;

END_IF 
{endregion}	
	 
{region "WorkFlow 2 -  CICLO DI RIPOSO"}
WF02_CicloDiRiposo();
{endregion}	 

{region "WorkFlow 3 -  CICLO PRELIEVO FALDA"}
WF03_CicloPrelFalda();
{endregion}	 

{region "WorkFlow 4 -  CICLO DEPOSITO FALDA"}		  
WF04_CicloDepFalda();
{endregion}	 

{region "WorkFlow 5 -  CICLO PRELIEVO LASTRA DA PP"}
WF05_CicloPrelLastraDaPP();
{endregion}	 

{region "WorkFlow 6 -  CICLO DEPOSITO LASTRA DA PP"}
WF06_CicloDepLastraDaPP();
{endregion}	 

{region "WorkFlow 7 -  CICLO PRELIEVO LASTRA DA WA"}
WF07_CicloPrelLastraDaWA();
{endregion}	 

{region "WorkFlow 8 -  CICLO DEPOSITO SU PAREGGIATORE "}
WF08_CicloDepLastraSuPareggiatore();
{endregion}	 
	 
{region "WorkFlow 9 -  CICLO DEPOSITO LASTRA DA WA"}
WF09_CicloDepLastraDaWA();
{endregion}	 

{region "WorkFlow 10 -  CICLO PRELIEVO LASTRA DA WA DEPAL"}
WF10_CicloPelLastra_Depal();
{endregion}	 	 

{region "WorkFlow 11 -  CICLO DEPOSITO FALDA DEPAL "}
WF11_CicloDepFalde_Depal();
{endregion}	 

{region "WorkFlow 12 -  CICLO DEPOSITO LASTRA DEPAL "}
WF12_CicloDepLastra_Depal();
{endregion}	 


(* Setto la memoria di richiesta stop in fase *)
WaitPositionRequest := (WaitPositionRequest OR ExternalWaitPositionRequest OR CmdExe.PhaseStopRequest > 0);

{region "GESTIONE INTERPOLAZIONE"}
(* Richiamo la FB di interpolazione degli assi *)
FROM_HMI_PAL.HMI_AbilitaInterpolazioneAssi := TRUE;
IF FROM_HMI_PAL.HMI_AbilitaInterpolazioneAssi THEN
	(* Se gli assi stanno accelerando o decelerando NON ESEGUO l'interpolazione *)
	IF (ProgrammaToModule_X.InterpolaAsse = INTERPOLAZIONE_ASSE AND (Modules^.AX_X.Ax^.AxRef^.Status.Accelerating OR Modules^.AX_X.Ax^.AxRef^.Status.Decelerating)) OR ProgrammaToModule_X.Stato <> DA_ESEGUIRE THEN
		ProgrammaToModule_X.InterpolaAsse := NO_INTERPOLAZIONE_ASSE;
	END_IF
	IF (ProgrammaToModule_Y.InterpolaAsse = INTERPOLAZIONE_ASSE AND (Modules^.AX_Y.Ax^.AxRef^.Status.Accelerating OR Modules^.AX_Y.Ax^.AxRef^.Status.Decelerating)) OR ProgrammaToModule_Y.Stato <> DA_ESEGUIRE THEN
		ProgrammaToModule_Y.InterpolaAsse := NO_INTERPOLAZIONE_ASSE;
	END_IF
	IF (ProgrammaToModule_Z.InterpolaAsse = INTERPOLAZIONE_ASSE AND (Modules^.AX_Z.Ax^.AxRef^.Status.Accelerating OR Modules^.AX_Z.Ax^.AxRef^.Status.Decelerating)) OR ProgrammaToModule_Z.Stato <> DA_ESEGUIRE THEN
		ProgrammaToModule_Z.InterpolaAsse := NO_INTERPOLAZIONE_ASSE;
	END_IF
	IF (ProgrammaToModule_J.InterpolaAsse = INTERPOLAZIONE_ASSE AND (Modules^.AX_J.Ax^.AxRef^.Status.Accelerating OR Modules^.AX_J.Ax^.AxRef^.Status.Decelerating)) OR ProgrammaToModule_J.Stato <> DA_ESEGUIRE THEN
		ProgrammaToModule_J.InterpolaAsse := NO_INTERPOLAZIONE_ASSE;
	END_IF
	
	Interpolazione_Assi(InterpolaAssi 	:=  ADR(STARTInterpolazioneASSI^), 			(* Abilitazione dell'interpolazione degli assi *)
						RitardoEsecuzione := RitardoEsecuzioneInterpolazione,
						TempoCompensazioneDec := TempoCompensazioneDecelerazione,
						TempCompensazioneAcc := TempoCompensazioneAccelerazione,
						AssiInterpolati := ADR(AssiInterpolati),					(* Variabile che indica se gli assi sono stati interpolati *)
						DeltaMinimoInterpolazione_X := 2,
						DeltaMinimoInterpolazione_Y := 2,
						DeltaMinimoInterpolazione_Z := 2,
						DeltaMinimoInterpolazione_J := 1,
						(* Abilitazione degli assi interpolati *)
						Interpola_X 	:= ADR(ProgrammaToModule_X.InterpolaAsse),		(* Se TRUE abilita l'interpolazione dell'asse X *)
						Interpola_Y 	:= ADR(ProgrammaToModule_Y.InterpolaAsse),		(* Se TRUE abilita l'interpolazione dell'asse Y *)
						Interpola_Z 	:= ADR(ProgrammaToModule_Z.InterpolaAsse),		(* Se TRUE abilita l'interpolazione dell'asse Z *)
						Interpola_J 	:= ADR(ProgrammaToModule_J.InterpolaAsse),		(* Se TRUE abilita l'interpolazione dell'asse J *)
						(* Quota di inizio Interpolazione *)
						PuntoIniziale_X := Modules^.AX_X.Ax^.AxRef^.NcToPlc.ActPos,	(* Punto di Partenza asse *)
						PuntoIniziale_Y := Modules^.AX_Y.Ax^.AxRef^.NcToPlc.ActPos,	(* Punto di Partenza asse *)
						PuntoIniziale_Z := Modules^.AX_Z.Ax^.AxRef^.NcToPlc.ActPos,	(* Punto di Partenza asse *)
						PuntoIniziale_J := Modules^.AX_J.Ax^.AxRef^.NcToPlc.ActPos,	(* Punto di Partenza asse *)
						(* Quota di destinazione *)
						PuntoFinale_X 	:= ProgrammaToModule_X.Quota_Destinazione,	(* Punto di Arrivo asse *)
						PuntoFinale_Y 	:= ProgrammaToModule_Y.Quota_Destinazione,	(* Punto di Arrivo asse *)
						PuntoFinale_Z 	:= ProgrammaToModule_Z.Quota_Destinazione,	(* Punto di Arrivo asse *)
						PuntoFinale_J 	:= ProgrammaToModule_J.Quota_Destinazione,	(* Punto di Arrivo asse *)
						(* Dinamica Asse X *)	
						Vel_MAX_X		:= ProgrammaToModule_X.Velocita,			(* Velocità MASSIMA dell'asse X *)
						Acc_MAX_X		:= ProgrammaToModule_X.Accelerazione,		(* Accelerazione MASSIMA Asse X *)
						Dec_MAX_X		:= ProgrammaToModule_X.Decelerazione,		(* Decelerazione MASSIMA Asse X *)
						Jerk_MAX_X		:= ProgrammaToModule_X.Jerk,				(* Jerk MASSIMO Asse X *)
						(* Dinamica Massima Y *)
						Vel_MAX_Y		:= ProgrammaToModule_Y.Velocita,			(* Velocità MASSIMA dell'asse Y *)
						Acc_MAX_Y		:= ProgrammaToModule_Y.Accelerazione,		(* Accelerazione MASSIMA Asse Y *)
						Dec_MAX_Y		:= ProgrammaToModule_Y.Decelerazione,		(* Decelerazione MASSIMA Asse Y *)
						Jerk_MAX_Y		:= ProgrammaToModule_Y.Jerk,				(* Jerk MASSIMO Asse Y *)
						(* Dinamica Massima Z *)
						Vel_MAX_Z		:= ProgrammaToModule_Z.Velocita,			(* Velocità MASSIMA dell'asse Z *)
						Acc_MAX_Z		:= ProgrammaToModule_Z.Accelerazione,		(* Accelerazione MASSIMA Asse Z *)
						Dec_MAX_Z		:= ProgrammaToModule_Z.Decelerazione,		(* Decelerazione MASSIMA Asse Z *)
						Jerk_MAX_Z		:= ProgrammaToModule_Z.Jerk,				(* Jerk MASSIMO Asse Z *)
						(* Dinamica Massima Asse J *)
						Vel_MAX_J		:= ProgrammaToModule_J.Velocita,			(* Velocità MASSIMA dell'asse J *)
						Acc_MAX_J		:= ProgrammaToModule_J.Accelerazione,		(* Accelerazione MASSIMA Asse J *)
						Dec_MAX_J		:= ProgrammaToModule_J.Decelerazione,		(* Decelerazione MASSIMA Asse J *)
						Jerk_MAX_J		:= ProgrammaToModule_J.Jerk,				(* Jerk MASSIMO Asse J *)
						(* Accelerazione iniziale degli assi *)
						Acc_Iniziale_X  := ABS(Modules^.AX_X.Ax^.AxRef^.NcToPlc.SetAcc), 
						Acc_Iniziale_Y  := ABS(Modules^.AX_Y.Ax^.AxRef^.NcToPlc.SetAcc), 
						Acc_Iniziale_Z  := ABS(Modules^.AX_Z.Ax^.AxRef^.NcToPlc.SetAcc), 
						Acc_Iniziale_J  := ABS(Modules^.AX_J.Ax^.AxRef^.NcToPlc.SetAcc), 
						(* Velocità iniziale degli assi *)
						Vel_Iniziale_X	:= ABS(Modules^.AX_X.Ax^.AxRef^.NcToPlc.SetVelo),
						Vel_Iniziale_Y	:= ABS(Modules^.AX_Y.Ax^.AxRef^.NcToPlc.SetVelo),
						Vel_Iniziale_Z	:= ABS(Modules^.AX_Z.Ax^.AxRef^.NcToPlc.SetVelo),
						Vel_Iniziale_J	:= ABS(Modules^.AX_J.Ax^.AxRef^.NcToPlc.SetVelo),
						(* Set della velocità di percorrenza e del tempo di accelerazione/decelerazione *)
						Vel_Percorso	:= MAX(1000,FROM_HMI_PAL.HMI_VelocitaPercorso),		(* Velocità di percorenza della traiettoria interpolata *)
						TAcc			:= MIN(10,FROM_HMI_PAL.HMI_TempoAccDec));		      	    (* Tempo di accelerazione *)
						
						IF AssiInterpolati THEN
							IF ProgrammaToModule_X.InterpolaAsse = INTERPOLAZIONE_ASSE THEN
								ProgrammaToModule_X.Velocita 		:= Interpolazione_Assi.Vel_X;		
								ProgrammaToModule_X.Accelerazione 	:= MAX(10,Interpolazione_Assi.Acc_OUT_X);	
								ProgrammaToModule_X.Decelerazione 	:= MAX(10,Interpolazione_Assi.Dec_OUT_X);
								ProgrammaToModule_X.Jerk 			:= ProgrammaToModule_X.Jerk;//5000;//Interpolazione_Assi.Jerk_OUT_X;
							ELSE
								ProgrammaToModule_X.Jerk			:= ProgrammaToModule_X.Jerk; 				
							END_IF
		
							IF ProgrammaToModule_Y.InterpolaAsse = INTERPOLAZIONE_ASSE THEN //
								ProgrammaToModule_Y.Velocita 		:= Interpolazione_Assi.Vel_Y;	
								ProgrammaToModule_Y.Accelerazione 	:= MAX(10,Interpolazione_Assi.Acc_OUT_Y);
								ProgrammaToModule_Y.Decelerazione 	:= MAX(10,Interpolazione_Assi.Dec_OUT_Y);	
								ProgrammaToModule_Y.Jerk 			:= ProgrammaToModule_Y.Jerk;//5000;//Interpolazione_Assi.Jerk_OUT_Y;
							ELSE
								ProgrammaToModule_Y.Jerk			:= ProgrammaToModule_Y.Jerk;
							END_IF	
								
							IF ProgrammaToModule_Z.InterpolaAsse = INTERPOLAZIONE_ASSE THEN // 
								ProgrammaToModule_Z.Velocita 		:= Interpolazione_Assi.Vel_Z;		
								ProgrammaToModule_Z.Accelerazione 	:= MAX(10,Interpolazione_Assi.Acc_OUT_Z);		
								ProgrammaToModule_Z.Decelerazione 	:= MAX(10,Interpolazione_Assi.Dec_OUT_Z);		
								ProgrammaToModule_Z.Jerk 			:= ProgrammaToModule_J.Jerk;//5000;//Interpolazione_Assi.Jerk_OUT_Z;	
							ELSE
								ProgrammaToModule_Z.Jerk			:= ProgrammaToModule_J.Jerk;	
							END_IF
							 
							IF ProgrammaToModule_J.InterpolaAsse  = INTERPOLAZIONE_ASSE	 THEN 
								ProgrammaToModule_J.Velocita 		:= Interpolazione_Assi.Vel_J;
								ProgrammaToModule_J.Accelerazione 	:= MAX(1,Interpolazione_Assi.Acc_OUT_J);
								ProgrammaToModule_J.Decelerazione 	:= MAX(1,Interpolazione_Assi.Dec_OUT_J);
								ProgrammaToModule_J.Jerk			:= ProgrammaToModule_J.Jerk;//5000;//Interpolazione_Assi.Jerk_OUT_J;
							ELSE
								ProgrammaToModule_J.Jerk			:= ProgrammaToModule_J.Jerk;
							END_IF
						END_IF
			
END_IF

//ProgrammaToModule_X.Jerk			:= 1000000000000;
//ProgrammaToModule_Y.Jerk			:= 1000000000000;
//PRogrammaToModule_Z.Jerk			:= 1000000000000;
//ProgrammaToModule_J.Jerk			:= 1000000000000;
//ProgrammaToModule_K.Jerk			:= 1000000000000;
(* Sbianco i flag di richiesta interpolazione *)
IF AssiInterpolati THEN
	FOR IndiceForSb := 0 TO 200 DO
		Programma_X[IndiceForSb].InterpolaAsse := NO_INTERPOLAZIONE_ASSE;
		Programma_Y[IndiceForSb].InterpolaAsse := NO_INTERPOLAZIONE_ASSE;
		Programma_Z[IndiceForSb].InterpolaAsse := NO_INTERPOLAZIONE_ASSE;
		Programma_J[IndiceForSb].InterpolaAsse := NO_INTERPOLAZIONE_ASSE;	
	END_FOR
END_IF
{endregion}	

(* ******************************************************************************************************** *)
(* Handshakes *)
(* ******************************************************************************************************** *)
					
(* ******************************************************************************************************** *)
(* State Input/Output *)
(* ******************************************************************************************************** *)
(* Fill Input/Output bit with sensor, electrovalve, etc. status *)

(* ******************************************************************************************************** *)
(* Errors *)
(* ******************************************************************************************************** *)

(* ******************************************************************************************************** *)
(* Input *)
(* ******************************************************************************************************** *)
(*Azzeramento comando di step HMI*)
HMI_CommandSTEP := CommandSTEP;

(* ******************************************************************************************************** *)
(* Error Check - Clear All Output!!! *)
(* ******************************************************************************************************** *)
IF TFPalletizerIsModuleError(Modules) THEN
	IF CmdExe.Code <> CmdNOP THEN
		IF CmdExe.Code <> CmdSTOP AND
			CmdExe.Code <> CmdPOWER AND
			CmdExe.Code <> CmdRESET AND
			CmdExe.Code <> CmdINIT AND
			CmdExe.Code <> CmdMAN AND
			CmdExe.Code <> CmdCICLORIPOSO THEN
			TFCommandClear(ADR(CmdNext));
			TFCommandExeClear(ADR(CmdExe));
			(* Clear All Output Here *)

		END_IF
	END_IF
	//OUT.HomeDone := FALSE;
END_IF;

(* ******************************************************************************************************** *)
(* Error Check - All Modules *)
(* ******************************************************************************************************** *)

(* ******************************************************************************************************** *)
(* Alarm *)
(* ******************************************************************************************************** *)
IF NOT IN.SensorAir AND NOT AirAlarmTrig THEN
	AirAlarmTrig := TRUE;
	TFParametersArrayClear(ADR (ParametersArray));
	TFCommandSend(CmdSTOP,ParametersArray,Cmd);
	TFError(ErrMACHINEPALLETIZER_AIR,ErrNULL,ADR(CmdExe),ADR(State),ADR(Error),ADR(ErrorLog));
END_IF

IF NOT IN.Sensor24Volt AND NOT Volt24Trig THEN
	Volt24Trig := TRUE;
	TFParametersArrayClear(ADR (ParametersArray));
	TFCommandSend(CmdSTOP,ParametersArray,Cmd);
	TFError(ErrMACHINEPALLETIZER_MAIN24V,ErrNULL,ADR(CmdExe),ADR(State),ADR(Error),ADR(ErrorLog));
END_IF

(* Controllo dei sensori di sicurezza delle cinghie *)
IF NOT IN.Y_BeltSafety AND NOT BeltSafetyTRIG AND IN.Mode.Auto THEN
	BeltSafetyTRIG := TRUE;
	TFParametersArrayClear(ADR(ParametersArray));
	TFCommandSend(CmdSTOP,ParametersArray,Cmd);
	TFError(ErrYBELTSAFETY,ErrNULL,ADR(CmdExe),ADR(State),ADR(Error),ADR(ErrorLog));
END_IF

IF NOT IN.Z_BeltSafety AND NOT BeltSafetyTRIG AND IN.Mode.Auto THEN
	BeltSafetyTRIG := TRUE;
	TFParametersArrayClear(ADR(ParametersArray));
	TFCommandSend(CmdSTOP,ParametersArray,Cmd);
	TFError(ErrZBELTSAFETY,ErrNULL,ADR(CmdExe),ADR(State),ADR(Error),ADR(ErrorLog));
END_IF

(* Controllo comunicazione con Trasporti *)

TFTimerSet(ADR(TimerComTrasporti),2000,IN.WD_Trasporti);
IF TFTimerDone(ADR(TimerComTrasporti)) and AbilitaErroreComunicazioneTrasporti THEN
	TFError(ErrCOMUNICAZTRASPORTI,ErrNULL,ADR(CmdExe),ADR(State),ADR(Error),ADR(ErrorLog));
END_IF


(* ******************************************************************************************************** *)
(* Diagnostic State *)
(* ******************************************************************************************************** *)

(* ******************************************************************************************************** *)
(* Machine Horn/Error/Warning/Run Outputs *)
(* ******************************************************************************************************** *)
(* Warning/Error Lamp + Error Horn *)
w := 0;
e := 0;
(* Add Others Modules *)
//IF TFIsModuleWarning(Modules^.Robot.Warning) THEN w := w + 1; END_IF
//IF TFIsModuleError(Modules^.Robot.Error) THEN e := e + 1; END_IF

(* Stop Request in case of one or more Modules Error *)
IF e <> 0 THEN
	CmdExe.PhaseStopRequest := 1;
END_IF

OUT.Warning := MachinePalletizer_TF.CmdExe.Code = CmdDO AND 
				ActualPickingListFromHMI[1].State = e_StatoWorkOrder.TERMINATO AND 
				ActualPickingListFromHMI[2].State = e_StatoWorkOrder.TERMINATO AND 
				ActualPickingListFromHMI[3].State = e_StatoWorkOrder.TERMINATO AND 
				MachinePalletizer_TF.InWaitPosition;
				
OUT.Error := Modules^.AX_X.Error.Code > 0 OR
			 Modules^.AX_Y.Error.Code > 0 OR
			 Modules^.AX_Z.Error.Code > 0 OR
			 Modules^.AX_J.Error.Code > 0 OR
			 Modules^.Pinza.Error.Code > 0 OR
			 Error.Code > 0 OR 
			 LGVError > 0 OR
			 LayerStackEmpty > 0;

(* Controllo tastatori di sicurezza pinza, attivo il controllo SEMPRE quando macchina in automatico!!!! *)
IF MachinePalletizer_TF.IN.Mode.Auto THEN
	TouchErrorEnable := TRUE;
END_IF
IF TouchErrorEnable AND 
(Modules^.AX_X.Error.Code  = ErrTOUCHEMERGENCY OR
 Modules^.AX_Y.Error.Code = ErrTOUCHEMERGENCY OR
 Modules^.AX_Z.Error.Code = ErrTOUCHEMERGENCY OR
 Modules^.AX_J.Error.Code = ErrTOUCHEMERGENCY) THEN
 	TFError(ErrTOUCHEMERGENCY,ErrNULL,ADR(CmdExe),ADR(State),ADR(Error),ADR(ErrorLog));
	CmdExe.PhaseStopRequest := 1;
	CmdExe.RapidStopRequest := 1;
END_IF
			 
(* Errore generato all'interno del TFLGV*)
IF LGVError > 0 THEN
	TFError(LGVError,ErrNULL,ADR(CmdExe),ADR(State),ADR(Error),ADR(ErrorLog));
END_IF
(* Errore generato all'interno del TFLGV*)
IF GateAccessError > 0 THEN
	TFError(GateAccessError,ErrNULL,ADR(CmdExe),ADR(State),ADR(Error),ADR(ErrorLog));
END_IF

IF TFTimerDone(ADR(TimerLamp)) THEN
	TFTimerSet(ADR(TimerLamp),1000,TRUE);
	ClockLamp := NOT ClockLamp;
END_IF

IF (CmdExe.Code = CmdHOME OR CmdExe.Code = CmdDO) AND PalletStackEmpty = 0 AND LayerStackEmpty = 0 AND AllWABusy = 0 THEN
	OUT.Run := TRUE;
ELSIF (CmdExe.Code = CmdHOME OR CmdExe.Code = CmdDO) AND (PalletStackEmpty > 0 OR LayerStackEmpty > 0 OR AllWABusy > 0) THEN
	OUT.Run := ClockLamp;
ELSE
	OUT.Run := FALSE;	
END_IF	

IF IN.Mode.ResetRequest THEN
	HornAck := TRUE;
END_IF
IF TFTimerDone(ADR(Timer1000)) THEN
	TFTimerSet(ADR(Timer1000),1000,TRUE);
	HornClock := NOT HornClock;
	OUT.Horn := OUT.Error AND HornClock AND NOT HornAck;
	IF NOT OUT.Error THEN HornAck := FALSE; END_IF
END_IF

IF NOT MachinePalletizer_TF.IN.Mode.Auto AND AutoTrig THEN
	AutoToMan := TRUE;
END_IF
AutoTrig := MachinePalletizer_TF.IN.Mode.Auto;

IF GateAccesExecuted AND NOT GateAccesTrig THEN
	GateAcces := TRUE;
END_IF
GateAccesTrig := GateAccesExecuted;

IF IN.Mode.RapidStopRequest AND NOT ExecuteStopTilterTRIG THEN
	ExecuteStopTilter := TRUE;
END_IF
ExecuteStopTilterTRIG := IN.Mode.RapidStopRequest;

OUT.ClockSegnalazioni := HornClock;

// Clock Segnalazione Alternato
TFTimerCall(ADR(TimerONAlternato),Cfg.TimeBase);
TFTimerCall(ADR(TimerOFFAlternato),Cfg.TimeBase);

TFTimerSet(ADR(TimerONAlternato),300,NOT OUT.ClockSegnalazioniAlternato); //Tempo Sirena ON
TFTimerSet(ADR(TimerOFFAlternato),2000,OUT.ClockSegnalazioniAlternato); //Tempo Sirena OFF 

IF TFTimerDone(ADR(TimerOFFAlternato)) THEN
	OUT.ClockSegnalazioniAlternato := TRUE;
ELSIF TFTimerDone(ADR(TimerONAlternato)) THEN
	OUT.ClockSegnalazioniAlternato := FALSE;
END_IF

//AutoReset Sirena Segnalazioni
TFTimerCall(ADR(TimerSirenaOFF_Segnalazioni),Cfg.TimeBase);

TFTimerSet(ADR(TimerSirenaOFF_Segnalazioni),300000,NOT OUT.Warning); //Tempo dopo il quale la sirena smette di suonare

IF TFTimerDone(ADR(TimerSirenaOFF_Segnalazioni)) THEN
	OUT.ResetSirenaSegnalazioni := TRUE;
ELSIF AutoToMan THEN //se metto in manuale, resetto il timer
	OUT.ResetSirenaSegnalazioni := FALSE;	
END_IF


(* ******************************************************************************************************** *)
(* Common Outputs *)
(* ******************************************************************************************************** *)

ACTION WF02_CicloDiRiposo:
(*-------------------------------------------------------------------------------------------*)
(* WorkFlow 2 -  CICLO DI RIPOSO *)
(*-------------------------------------------------------------------------------------------*)
NumeroWF :=2;
IF WorkFlow[NumeroWF].Enable THEN

	IF NOT TFCommandCaseIsEnable(ADR(CmdExe)) THEN RETURN; END_IF
	CASE WorkFlow[NumeroWF].WFCase OF

		(* Case 0 *)
		0:  WorkFlow[NumeroWF].State := StateWF_RUN;
			STEPCicloDONE := FALSE;
			OUT.StartTilter := TRUE;
			TFWorkFlowCase(ADR(WorkFlow[NumeroWF]),1,WorkflowCase_INC);
	
		(* Case 1 - Chiamata del FB del ciclo di riposo per Valorizzarne i valori*)
		1:	IF CmdExe.RapidStopRequest > 0 OR
				TFPalletizerIsModuleError(Modules) OR Error.Code <> 0 THEN
					TFWorkFlowCase(ADR(WorkFlow[NumeroWF]),100,WorkflowCase_JMP);
			ELSE

				IF QuotaFuoriIngombro_X_AVUOTO = 0 THEN
					QuotaFuoriIngombro_X_AVUOTO := WorkPickPoint^[1].X;
				END_IF
				IF QuotaFuoriIngombro_Y_AVUOTO = 0 THEN
					QuotaFuoriIngombro_Y_AVUOTO := WorkPickPoint^[1].Y;
				END_IF
				IF QuotaFuoriIngombro_Z_AVUOTO = 0 THEN
					QuotaFuoriIngombro_Z_AVUOTO := WorkPickPoint^[1].Z + 300;
				END_IF
				//IF QuotaFuoriIngombro_J_AVUOTO = 0 THEN
				//	QuotaFuoriIngombro_J_AVUOTO := 90;
				//END_IF
				

				TFProgramma_Ciclo_Riposo.X_Par := ParametriProgramma_X_CicloRiposo;
				TFProgramma_Ciclo_Riposo.Y_Par := ParametriProgramma_Y_CicloRiposo;
				TFProgramma_Ciclo_Riposo.Z_Par := ParametriProgramma_Z_CicloRiposo;
				TFProgramma_Ciclo_Riposo.J_Par := ParametriProgramma_J_CicloRiposo;
				//TFProgramma_Ciclo_Riposo.K_Par := ParametriProgramma_K_CicloRiposo;
				(******************************************************************************)					 
				TFProgramma_Ciclo_Riposo.Quota_Riposo_X := Mission^.XPick;
				TFProgramma_Ciclo_Riposo.Quota_Riposo_Y := Mission^.YPick;
				TFProgramma_Ciclo_Riposo.Quota_Riposo_Z := Mission^.ZPick;
				TFProgramma_Ciclo_Riposo.Quota_Riposo_J := Mission^.JPick;
				(******************************************************************************)
				TFProgramma_Ciclo_Riposo.Quota_Fuori_Ingombro_X := QuotaFuoriIngombro_X_AVUOTO; 
				TFProgramma_Ciclo_Riposo.Quota_Fuori_Ingombro_Y := QuotaFuoriIngombro_Y_AVUOTO;
 				TFProgramma_Ciclo_Riposo.Quota_Fuori_Ingombro_Z := QuotaFuoriIngombro_Z_AVUOTO;
				TFProgramma_Ciclo_Riposo.Quota_Fuori_Ingombro_J := QuotaFuoriIngombro_J_AVUOTO;
				
				TFProgramma_Ciclo_Riposo();
				(* Valuto se è abilitata l'interpolazione degli assi *)
				IF NOT AbilitaInterpolazioneAssi^ THEN
					TFWorkFlowCase(ADR(WorkFlow[NumeroWF]),20,WorkflowCase_JMP);	// Case con FB SENZA interpolazione
				ELSE
					TFWorkFlowCase(ADR(WorkFlow[NumeroWF]),30,WorkflowCase_JMP);	// Case con FB CON interpolazione
				END_IF
			END_IF;
			
		(* Case 20 - Chiamata FB del ciclo di lavoro *)	
		20:	
			TFWorkFlowCase(ADR(WorkFlow[NumeroWF]),30,WorkflowCase_JMP);	// Case con FB CON interpolazione

		
		(* Case 30 - Chiamata FB del ciclo di lavoro *)	
		30:	
			IF CmdExe.RapidStopRequest > 0 OR
				TFPalletizerIsModuleError(Modules) OR Error.Code <> 0 THEN
					TFCiclo_Di_Riposo.InterrompiCiclo := TRUE;
			ELSE
				TFCiclo_Di_Riposo.InterrompiCiclo := FALSE;
			END_IF
			TFCiclo_Di_Riposo.Ciclo						:= ADR(Ciclo_Di_Riposo);
			TFCiclo_Di_Riposo.Programma					:= ADR(TFProgramma_Ciclo_Riposo);
			TFCiclo_Di_Riposo.ModuleAX_X 				:= ADR(Modules^.AX_X);
			TFCiclo_Di_Riposo.ModuleAX_Y 				:= ADR(Modules^.AX_Y);
			TFCiclo_Di_Riposo.ModuleAX_Z 				:= ADR(Modules^.AX_Z);
			TFCiclo_Di_Riposo.ModuleAX_J 				:= ADR(Modules^.AX_J);
			TFCiclo_Di_Riposo.ModulePinza 		:= ADR(Modules^.Pinza);
			TFCiclo_Di_Riposo.StartInterpolazioneAssi 		:= ADR(STARTInterpolazioneASSI^);
			TFCiclo_Di_Riposo.AbilitazioneGlobalePassMode 		:= Traiettoria^.PassModeGlobalEnable;
			TFCiclo_Di_Riposo.Abilita_Ciclo_Step		:= AbilitazioCiclo_TEST_STEP;
			
			IF CommandSTEP AND NOT CommandSTEPTRIG THEN
				TFCiclo_Di_Riposo.Command_Step	:= TRUE;
				CommandSTEPTRIG := TRUE;
			ELSIF NOT CommandSTEP AND NOT CommandSTEPTRIG THEN
				TFCiclo_Di_Riposo.Command_Step	:= FALSE;
				CommandSTEPTRIG := FALSE;
				CommandSTEP := FALSE;
			ELSIF  STEPCicloDONE THEN
				TFCiclo_Di_Riposo.Command_Step	:= FALSE;
				CommandSTEP := FALSE;
				CommandSTEPTRIG := FALSE;
			END_IF
			TFCiclo_Di_Riposo();
			STEPCicloDONE := TFCiclo_Di_Riposo.STEPDone;
			
			IF TFCiclo_Di_Riposo.Ciclo^.Stato = TERMINATO THEN
				TFWorkFlowCase(ADR(WorkFlow[NumeroWF]),100,WorkflowCase_JMP);
			ELSIF TFCiclo_Di_Riposo.Errore > 0 THEN
				TFError(TFCiclo_Di_Riposo.Errore,ErrNULL,ADR(CmdExe),ADR(State),ADR(Error),ADR(ErrorLog));	
				TFWorkFlowCase(ADR(WorkFlow[NumeroWF]),999,WorkflowCase_JMP);	 
			ELSIF TFCiclo_Di_Riposo.Ciclo^.Stato = INTERROTTO THEN	
				TFWorkFlowCase(ADR(WorkFlow[NumeroWF]),999,WorkflowCase_JMP);		
			END_IF

		(* Case 100 *)
		100:WorkFlow[NumeroWF].State := StateWF_END;
			WorkFlow[NumeroWF].Enable := FALSE;
			CommandSTEP := FALSE;
			CommandSTEPTRIG := FALSE;
			AssiInterpolati := FALSE;

		(* Case 999 *)
		(* WorkFlow ERROR *)
		StateWF_ERROR:
			TFWorkFlowError(ADR(WorkFlow[NumeroWF]),ADR(WorkFlowErrorLog[NumeroWF]));
			CmdExe.PhaseStopRequest := 1;
			CmdExe.RapidStopRequest := 1;
			WorkFlow[NumeroWF].Enable := FALSE;
			CommandSTEP := FALSE;
			CommandSTEPTRIG := FALSE;
			AssiInterpolati := FALSE;
		
		ELSE						
			TFWorkFlowError(ADR(WorkFlow[NumeroWF]),ADR(WorkFlowErrorLog[NumeroWF]));
			TFError(ErrNOCMDCASE,ErrNULL,ADR(CmdExe),ADR(State),ADR(Error),ADR(ErrorLog));
		
	END_CASE;
	
END_IF
END_ACTION

ACTION WF03_CicloPrelFalda:
(*-------------------------------------------------------------------------------------------*)
(* WorkFlow 3 -  CICLO PRELIEVO FALDA *)
(*-------------------------------------------------------------------------------------------*)		
NumeroWF:=3;	
IF WorkFlow[NumeroWF].Enable THEN

	IF NOT TFCommandCaseIsEnable(ADR(CmdExe)) THEN RETURN; END_IF
	CASE WorkFlow[NumeroWF].WFCase OF

		(* Case 0 *)
		0:  WorkFlow[NumeroWF].State := StateWF_RUN;
			STEPCicloDONE := FALSE;
			OUT.StartTilter := FALSE;
			TFWorkFlowCase(ADR(WorkFlow[NumeroWF]),1,WorkflowCase_INC);
	
		(* Case 1 - Chiamata del FB del ciclo di riposo per Valorizzarne i valori*)
		1:	IF CmdExe.RapidStopRequest > 0 OR
				TFPalletizerIsModuleError(Modules) THEN
					TFWorkFlowCase(ADR(WorkFlow[NumeroWF]),100,WorkflowCase_JMP);
			ELSE
				TFProgramma_Ciclo_Falda.X_Par := ParametriProgramma_X_CicloFalda;
				TFProgramma_Ciclo_Falda.Y_Par := ParametriProgramma_Y_CicloFalda;
				TFProgramma_Ciclo_Falda.Z_Par := ParametriProgramma_Z_CicloFalda;
				TFProgramma_Ciclo_Falda.J_Par := ParametriProgramma_J_CicloFalda;
				//TFProgramma_Ciclo_Falda.K_Par := ParametriProgramma_K_CicloFalda;
				
				(*X*)
				TFProgramma_Ciclo_Falda.Quota_Prelievo_Falda_X 					:= Traiettoria^.StartPoint.X;
				TFProgramma_Ciclo_Falda.Quota_Deposito_Falda_SuCatastaPallet_X 	:= Traiettoria^.EndPoint.X;
				TFProgramma_Ciclo_Falda.Quota_Deposito_Falda_SuPiazzola_X	 	:= Traiettoria^.EndPoint.X;	
				
				(*Y*)
				TFProgramma_Ciclo_Falda.Quota_Prelievo_Falda_Y 					:= Traiettoria^.StartPoint.Y;
				TFProgramma_Ciclo_Falda.Quota_Deposito_Falda_SuCatastaPallet_Y 	:= Traiettoria^.EndPoint.Y;
				TFProgramma_Ciclo_Falda.Quota_Deposito_Falda_SuPiazzola_Y		:= Traiettoria^.EndPoint.Y;
				TFProgramma_Ciclo_Falda.Quota_Fuori_Ingombro_Y 					:= QuotaFuoriIngombroColonne_Y;//(WorkSpace^.Y - IngombroSuperficialePinzaMAX_Global/2);
				
				(*Z*)
				TFProgramma_Ciclo_Falda.Quota_StartLenta_Prelievo_Falda_Z 					:= Traiettoria^.PuntoDiApproccioStartPoint.Z;
				TFProgramma_Ciclo_Falda.Quota_Prelievo_Falda_Z 								:= Traiettoria^.StartPoint.Z;
				TFProgramma_Ciclo_Falda.Quota_StartLenta_Deposito_Falda_SuPiazzola_Z 		:= Traiettoria^.PuntoDiApproccioEndPoint.Z;
				TFProgramma_Ciclo_Falda.Quota_Deposito_Falda_SuPiazzola_Z					:= Traiettoria^.EndPoint.Z;
				TFProgramma_Ciclo_Falda.Quota_StartLenta_Deposito_Falda_SuCatastaPallet_Z	:= Traiettoria^.PuntoDiApproccioEndPoint.Z;
				TFProgramma_Ciclo_Falda.Quota_Deposito_Falda_SuCatastaPallet_Z				:= Traiettoria^.EndPoint.Z;
				TFProgramma_Ciclo_Falda.QUota_Fuori_Ingombro_Falda_Z 						:= QuotaFuoriIngombro_Z_ConFALDA;
				TFProgramma_Ciclo_Falda.Quota_Attesa_Caduta_Falda_Z							:= Modules^.AX_Z.Ax^.Status.ActPosition + OffsetCadutaFalda;//Quota_Attesa_Caduta_Falda_Z;
								
				(*J*)
				TFProgramma_Ciclo_Falda.Quota_Rotazione_Prelievo_Falda 			:= Traiettoria^.StartPoint.J;
				TFProgramma_Ciclo_Falda.Quota_Rotazione_Deposito_Falda 			:= Traiettoria^.EndPoint.J;
				TFProgramma_Ciclo_Falda();
				(* Valuto se è abilitata l'interpolazione degli assi *)
				IF NOT AbilitaInterpolazioneAssi^ THEN
					TFWorkFlowCase(ADR(WorkFlow[NumeroWF]),20,WorkflowCase_JMP);	// Case con FB SENZA interpolazione
				ELSE
					TFWorkFlowCase(ADR(WorkFlow[NumeroWF]),30,WorkflowCase_JMP);	// Case con FB CON interpolazione
				END_IF
			END_IF;
			
		(* Case 20 - Chiamata FB del ciclo di lavoro *)	
		20:	
			TFWorkFlowCase(ADR(WorkFlow[3]),30,WorkflowCase_JMP);	// Case con FB CON interpolazione

			
		(* Case 30 - Chiamata FB del ciclo di lavoro *)	
		30:	
			IF CmdExe.RapidStopRequest > 0 OR
				TFPalletizerIsModuleError(Modules) THEN
					TFCiclo_Prelievo_Falda.InterrompiCiclo := TRUE;
			ELSE
				TFCiclo_Prelievo_Falda.InterrompiCiclo := FALSE;
			END_IF
			TFCiclo_Prelievo_Falda.Ciclo					:= ADR(Ciclo_Pelievo_Falda);
			TFCiclo_Prelievo_Falda.Programma				:= ADR(TFProgramma_Ciclo_Falda);
			TFCiclo_Prelievo_Falda.ModuleAX_X 				:= ADR(Modules^.AX_X);
			TFCiclo_Prelievo_Falda.ModuleAX_Y 				:= ADR(Modules^.AX_Y);
			TFCiclo_Prelievo_Falda.ModuleAX_Z 				:= ADR(Modules^.AX_Z);
			TFCiclo_Prelievo_Falda.ModuleAX_J 				:= ADR(Modules^.AX_J);
			TFCiclo_Prelievo_Falda.ModulePinza 		:= ADR(Modules^.Pinza);
			TFCiclo_Prelievo_Falda.StartInterpolazioneAssi 	:= ADR(STARTInterpolazioneASSI^);
			TFCiclo_Prelievo_Falda.AbilitazioneGlobalePassMode 		:= Traiettoria^.PassModeGlobalEnable;
			TFCiclo_Prelievo_Falda.Abilita_Ciclo_Step		:= AbilitazioCiclo_TEST_STEP;
			
			IF CommandSTEP AND NOT CommandSTEPTRIG THEN
				TFCiclo_Prelievo_Falda.Command_Step	:= TRUE;
				CommandSTEPTRIG := TRUE;
			ELSIF NOT CommandSTEP AND NOT CommandSTEPTRIG THEN
				TFCiclo_Prelievo_Falda.Command_Step	:= FALSE;
				CommandSTEPTRIG := FALSE;
				CommandSTEP := FALSE;
			ELSIF  STEPCicloDONE THEN
				TFCiclo_Prelievo_Falda.Command_Step	:= FALSE;
				CommandSTEP := FALSE;
				CommandSTEPTRIG := FALSE;
			END_IF
			
			TFCiclo_Prelievo_Falda();
			STEPCicloDONE := TFCiclo_Prelievo_Falda.STEPDone;
			
			IF Ciclo_Pelievo_Falda.Stato = TERMINATO THEN
				ProductOnGripper := KPRODUCTLOADED;
				TFWorkFlowCase(ADR(WorkFlow[NumeroWF]),100,WorkflowCase_JMP);
			ELSIF Ciclo_Pelievo_Falda.Stato = INTERROTTO THEN	
				TFWorkFlowCase(ADR(WorkFlow[NumeroWF]),999,WorkflowCase_JMP);		
			END_IF

		(* Case 100 *)
		100:WorkFlow[NumeroWF].State := StateWF_END;
			WorkFlow[NumeroWF].Enable := FALSE;
			CommandSTEP := FALSE;
			CommandSTEPTRIG := FALSE;
			AssiInterpolati := FALSE;

		(* Case 999 *)
		(* WorkFlow ERROR *)
		StateWF_ERROR:
			TFWorkFlowError(ADR(WorkFlow[NumeroWF]),ADR(WorkFlowErrorLog[5]));
			CmdExe.PhaseStopRequest := 1;
			CmdExe.RapidStopRequest := 1;
			WorkFlow[NumeroWF].Enable := FALSE;
			CommandSTEP := FALSE;
			CommandSTEPTRIG := FALSE;
			AssiInterpolati := FALSE;
				
		ELSE						
			TFWorkFlowError(ADR(WorkFlow[NumeroWF]),ADR(WorkFlowErrorLog[5]));
			TFError(ErrNOCMDCASE,ErrNULL,ADR(CmdExe),ADR(State),ADR(Error),ADR(ErrorLog));
		
	END_CASE;
	
END_IF
END_ACTION

ACTION WF04_CicloDepFalda:
(*-------------------------------------------------------------------------------------------*)
(* WorkFlow 4 -  CICLO DEPOSITO FALDA *)
(*-------------------------------------------------------------------------------------------*)	
NumeroWF:=4;	
IF WorkFlow[NumeroWF].Enable THEN

	IF NOT TFCommandCaseIsEnable(ADR(CmdExe)) THEN RETURN; END_IF
	CASE WorkFlow[NumeroWF].WFCase OF

		(* Case 0 *)
		0:  WorkFlow[NumeroWF].State := StateWF_RUN;
			STEPCicloDONE := FALSE;
			OUT.StartTilter := FALSE;
			TFWorkFlowCase(ADR(WorkFlow[NumeroWF]),1,WorkflowCase_INC);
	
		(* Case 1 - Chiamata del FB del ciclo di riposo per Valorizzarne i valori*)
		1:	IF CmdExe.RapidStopRequest > 0 OR
				TFPalletizerIsModuleError(Modules) THEN
				TFWorkFlowCase(ADR(WorkFlow[NumeroWF]),100,WorkflowCase_JMP);
			ELSE
				TFProgramma_Ciclo_Falda.X_Par := ParametriProgramma_X_CicloFalda;
				TFProgramma_Ciclo_Falda.Y_Par := ParametriProgramma_Y_CicloFalda;
				TFProgramma_Ciclo_Falda.Z_Par := ParametriProgramma_Z_CicloFalda;
				TFProgramma_Ciclo_Falda.J_Par := ParametriProgramma_J_CicloFalda;
				
				(*X*)
				TFProgramma_Ciclo_Falda.Quota_Prelievo_Falda_X 					:= Traiettoria^.StartPoint.X;
				TFProgramma_Ciclo_Falda.Quota_Deposito_Falda_SuCatastaPallet_X 	:= Traiettoria^.EndPoint.X;
				TFProgramma_Ciclo_Falda.Quota_Deposito_Falda_SuPiazzola_X	 	:= Traiettoria^.EndPoint.X;	
				
				(*Y*)
				TFProgramma_Ciclo_Falda.Quota_Prelievo_Falda_Y 					:= Traiettoria^.StartPoint.Y;
				TFProgramma_Ciclo_Falda.Quota_Deposito_Falda_SuCatastaPallet_Y 	:= Traiettoria^.EndPoint.Y;
				TFProgramma_Ciclo_Falda.Quota_Deposito_Falda_SuPiazzola_Y		:= Traiettoria^.EndPoint.Y;
				TFProgramma_Ciclo_Falda.Quota_Fuori_Ingombro_Y 					:= QuotaFuoriIngombroColonne_Y;//(WorkSpace^.Y - IngombroSuperficialePinzaMAX_Global/2);

				(*Z*)
				TFProgramma_Ciclo_Falda.Quota_StartLenta_Prelievo_Falda_Z 					:= Traiettoria^.PuntoDiApproccioStartPoint.Z;
				TFProgramma_Ciclo_Falda.Quota_Prelievo_Falda_Z 								:= Traiettoria^.StartPoint.Z;
				TFProgramma_Ciclo_Falda.Quota_StartLenta_Deposito_Falda_SuPiazzola_Z 		:= Traiettoria^.PuntoDiApproccioEndPoint.Z;
				TFProgramma_Ciclo_Falda.Quota_Deposito_Falda_SuPiazzola_Z					:= Traiettoria^.EndPoint.Z;
				TFProgramma_Ciclo_Falda.Quota_StartLenta_Deposito_Falda_SuCatastaPallet_Z	:= Traiettoria^.PuntoDiApproccioEndPoint.Z;
				TFProgramma_Ciclo_Falda.Quota_Deposito_Falda_SuCatastaPallet_Z				:= Traiettoria^.EndPoint.Z;
				TFProgramma_Ciclo_Falda.QUota_Fuori_Ingombro_Falda_Z 						:= QuotaFuoriIngombro_Z_ConFALDA;
				TFProgramma_Ciclo_Falda.Quota_Attesa_Caduta_Falda_Z							:= Modules^.AX_Z.Ax^.Status.ActPosition + OffsetCadutaFalda;//Quota_Attesa_Caduta_Falda_Z;
					
				(*J*)
				TFProgramma_Ciclo_Falda.Quota_Rotazione_Prelievo_Falda 			:= Traiettoria^.StartPoint.J;
				TFProgramma_Ciclo_Falda.Quota_Rotazione_Deposito_Falda 			:= Traiettoria^.EndPoint.J;
				TFProgramma_Ciclo_Falda();
				(* Valuto se è abilitata l'interpolazione degli assi *)
				IF NOT AbilitaInterpolazioneAssi^ THEN
					TFWorkFlowCase(ADR(WorkFlow[NumeroWF]),20,WorkflowCase_JMP);	// Case con FB SENZA interpolazione
				ELSE
					TFWorkFlowCase(ADR(WorkFlow[NumeroWF]),30,WorkflowCase_JMP);	// Case con FB CON interpolazione
				END_IF
			END_IF;
		(* Case 20 - Chiamata FB del ciclo di lavoro *)	
		20:	
			TFWorkFlowCase(ADR(WorkFlow[NumeroWF]),30,WorkflowCase_JMP);	// Case con FB CON interpolazione

			
		(* Case 30 - Chiamata FB del ciclo di lavoro *)	
		30:	
			IF CmdExe.RapidStopRequest > 0 OR
				TFPalletizerIsModuleError(Modules) THEN
				TFCiclo_Deposito_Falda.InterrompiCiclo := TRUE;
			ELSE
				TFCiclo_Deposito_Falda.InterrompiCiclo := FALSE;
			END_IF
			TFCiclo_Deposito_Falda.Ciclo					:= ADR(Ciclo_Deposito_Falda);
			TFCiclo_Deposito_Falda.Programma				:= ADR(TFProgramma_Ciclo_Falda);
			TFCiclo_Deposito_Falda.ModuleAX_X 				:= ADR(Modules^.AX_X);
			TFCiclo_Deposito_Falda.ModuleAX_Y 				:= ADR(Modules^.AX_Y);
			TFCiclo_Deposito_Falda.ModuleAX_Z 				:= ADR(Modules^.AX_Z);
			TFCiclo_Deposito_Falda.ModuleAX_J 				:= ADR(Modules^.AX_J);
			TFCiclo_Deposito_Falda.ModulePinza 		:= ADR(Modules^.Pinza);
			TFCiclo_Deposito_Falda.StartInterpolazioneAssi 	:= ADR(STARTInterpolazioneASSI^);
			TFCiclo_Deposito_Falda.AbilitazioneGlobalePassMode 		:= Traiettoria^.PassModeGlobalEnable;
			TFCiclo_Deposito_Falda.Abilita_Ciclo_Step		:= AbilitazioCiclo_TEST_STEP;
			(* Set della tipologia di deposito *)
			IF Workarea^[Mission^.PPlace].Typology = TYPOLOGY_STACK THEN 
				TFCiclo_Deposito_Falda.TipoDiDeposito		:= DEPOSITO_FALDA_SU_CATASTA;
			ELSIF Workarea^[Mission^.PPlace].Typology = TYPOLOGY_PALLET THEN
				TFCiclo_Deposito_Falda.TipoDiDeposito		:= DEPOSITO_FALDA_SU_PIAZZOLA;
			ELSE
				; //non dovrebbe mai accadere
			END_IF
			
			IF CommandSTEP AND NOT CommandSTEPTRIG THEN
				TFCiclo_Deposito_Falda.Command_Step	:= TRUE;
				CommandSTEPTRIG := TRUE;
			ELSIF NOT CommandSTEP AND NOT CommandSTEPTRIG THEN
				TFCiclo_Deposito_Falda.Command_Step	:= FALSE;
				CommandSTEPTRIG := FALSE;
				CommandSTEP := FALSE;
			ELSIF  STEPCicloDONE THEN
				TFCiclo_Deposito_Falda.Command_Step	:= FALSE;
				CommandSTEP := FALSE;
				CommandSTEPTRIG := FALSE;
			END_IF
			
			TFCiclo_Deposito_Falda();
			STEPCicloDONE := TFCiclo_Deposito_Falda.STEPDone;
			
			IF Ciclo_Deposito_Falda.Stato = TERMINATO THEN
				OUT.StartTilter := TRUE;
				ProductOnGripper := KNOPRODUCT;
				TFWorkFlowCase(ADR(WorkFlow[NumeroWF]),100,WorkflowCase_JMP);
			ELSIF Ciclo_Deposito_Falda.Stato = INTERROTTO THEN	
				TFWorkFlowCase(ADR(WorkFlow[NumeroWF]),999,WorkflowCase_JMP);		
			END_IF

		(* Case 100 *)
		100:WorkFlow[NumeroWF].State := StateWF_END;
			WorkFlow[NumeroWF].Enable := FALSE;
			CommandSTEP := FALSE;
			CommandSTEPTRIG := FALSE;
			TFWorkFlowCase(ADR(WorkFlow[NumeroWF]),0,WorkflowCase_JMP);
			AssiInterpolati := FALSE;

		(* Case 999 *)
		(* WorkFlow ERROR *)
		StateWF_ERROR:
			TFWorkFlowError(ADR(WorkFlow[NumeroWF]),ADR(WorkFlowErrorLog[NumeroWF]));
			CmdExe.PhaseStopRequest := 1;
			CmdExe.RapidStopRequest := 1;
			WorkFlow[NumeroWF].Enable := FALSE;
			CommandSTEP := FALSE;
			CommandSTEPTRIG := FALSE;
			AssiInterpolati := FALSE;
		
		ELSE						
			TFWorkFlowError(ADR(WorkFlow[NumeroWF]),ADR(WorkFlowErrorLog[NumeroWF]));
			TFError(ErrNOCMDCASE,ErrNULL,ADR(CmdExe),ADR(State),ADR(Error),ADR(ErrorLog));
		
	END_CASE;
	
END_IF
END_ACTION

ACTION WF05_CicloPrelLastraDaPP:
(*-------------------------------------------------------------------------------------------*)
(* WorkFlow 5 -  CICLO PRELIEVO LASTRA DA PP *)
(*-------------------------------------------------------------------------------------------*)	
NumeroWF := 5;	
IF WorkFlow[NumeroWF].Enable THEN

	IF NOT TFCommandCaseIsEnable(ADR(CmdExe)) THEN RETURN; END_IF
	CASE WorkFlow[NumeroWF].WFCase OF

		(* Case 0 *)
		0:  WorkFlow[NumeroWF].State := StateWF_RUN;
			STEPCicloDONE := FALSE;	
			OUT.StartTilter := TRUE;
			TFWorkFlowCase(ADR(WorkFlow[NumeroWF]),1,WorkflowCase_INC);
	
		(* Case 1 - Chiamata del FB del ciclo di riposo per Valorizzarne i valori*)
		1:	IF CmdExe.RapidStopRequest > 0  OR
				TFPalletizerIsModuleError(Modules) THEN
				TFWorkFlowCase(ADR(WorkFlow[NumeroWF]),100,WorkflowCase_JMP);
			ELSE

				TFProgramma_Ciclo_Lastra.X_Par := ParametriProgramma_X_CicloLastra;
				TFProgramma_Ciclo_Lastra.Y_Par := ParametriProgramma_Y_CicloLastra;
				TFProgramma_Ciclo_Lastra.Z_Par := ParametriProgramma_Z_CicloLastra;
				TFProgramma_Ciclo_Lastra.J_Par := ParametriProgramma_J_CicloLastra;
				
				(*X*)
				TFProgramma_Ciclo_Lastra.Quota_StartLenta_Prelievo_Lastra_X			:= Traiettoria^.PuntoDiApproccioStartPoint.X;
				TFProgramma_Ciclo_Lastra.Quota_Prelievo_Lastra_X 					:= Traiettoria^.StartPoint.X;
				TFProgramma_Ciclo_Lastra.Quota_StartLenta_Deposito_Lastra_X	 		:= Traiettoria^.PuntoDiApproccioEndPoint.X;	
				TFProgramma_Ciclo_Lastra.Quota_Deposito_Lastra_X 					:= Traiettoria^.EndPoint.X;
				TFProgramma_Ciclo_Lastra.Quota_Fuori_Ingombro_SenzaCarico_X			:= Traiettoria^.EndPoint.X;//STESSA QUOTA DI DEPOSITO X DEPAL UNIVERSAL
				TFProgramma_Ciclo_Lastra.Quota_Fuori_Ingombro_Carico_X				:= Traiettoria^.EndPoint.X;//STESSA QUOTA DI DEPOSITO X DEPAL UNIVERSAL
				
				(*Y*)
				TFProgramma_Ciclo_Lastra.Quota_StartLenta_Prelievo_Lastra_Y         := Traiettoria^.PuntoDiApproccioStartPoint.Y;;
				TFProgramma_Ciclo_Lastra.Quota_Prelievo_Lastra_Y 					:= Traiettoria^.StartPoint.Y;
				TFProgramma_Ciclo_Lastra.Quota_Distacco_Lastra_Y					:= Traiettoria^.PuntoDiPostPosizionamentoStartPoint.Y;
				TFProgramma_Ciclo_Lastra.Quota_StartLenta_Deposito_Lastra_Y			:= Traiettoria^.PuntoDiApproccioEndPoint.Y;
				TFProgramma_Ciclo_Lastra.Quota_Deposito_Lastra_Y 					:= Traiettoria^.EndPoint.Y;
				TFProgramma_Ciclo_Lastra.Quota_Fuori_Ingombro_Y 					:= QuotaFuoriIngombro_Y_AVUOTO;//DEVE ESSERE GUALE A QUELLE DEL CORRIDOIO
				
				(*Z*)
				TFProgramma_Ciclo_Lastra.Quota_StartLenta_Prelievo_Lastra_Z 		:= MAX(Traiettoria^.PuntoDiApproccioStartPoint.Z,AxisPar_Z.MinPosition);
				TFProgramma_Ciclo_Lastra.Quota_Prelievo_Lastra_Z 					:= MAX(Traiettoria^.StartPoint.Z,AxisPar_Z.MinPosition);
				TFProgramma_Ciclo_Lastra.Quota_StartLenta_Deposito_Lastra_Z			:= Traiettoria^.PuntoDiApproccioEndPoint.Z;
				IF HMI_AbilitaDepositoPaccoOrrizzontaleConTasteggio THEN
					TFProgramma_Ciclo_Lastra.Quota_Deposito_Lastra_Z					:= Traiettoria^.EndPoint.Z -100;
				ELSE
					TFProgramma_Ciclo_Lastra.Quota_Deposito_Lastra_Z					:= Traiettoria^.EndPoint.Z;
				END_IF
				TFProgramma_Ciclo_Lastra.Quota_Fuori_Ingombro_ConCarico_Z			:= QuotaFuoriIngombro_Z_ConPEZZO;
				TFProgramma_Ciclo_Lastra.Quota_Fuori_Ingombro_SenzaCarico_Z			:= QuotaFuoriIngombro_Z_AVUOTO;
				TFProgramma_Ciclo_Lastra.Quota_Distacco_Lastra_Z					:= Traiettoria^.PuntoDiPostPosizionamentoStartPoint.Z;
				TFProgramma_Ciclo_Lastra.Quota_PostScarico							:= Z_Riposo;	
			
				(*J*)
				TFProgramma_Ciclo_Lastra.Quota_Rotazione_Prelievo_Lastra 			:= Traiettoria^.StartPoint.J;
				TFProgramma_Ciclo_Lastra.Quota_Rotazione_Deposito_Lastra 			:= Traiettoria^.EndPoint.J;
				TFProgramma_Ciclo_Lastra.Quota_Rotazione_StartTasteggio_Lastra		:= Traiettoria^.StartPoint.J;
				TFProgramma_Ciclo_Lastra.Quota_Fuori_Ingombro_J						:= QuotaFuoriIngombro_J_AVUOTO;
				TFProgramma_Ciclo_Lastra.Quota_Rotazione_Sfogliatura 				:= Traiettoria^.StartPoint.J + HMI_GradiSfogliaturaJ;

				TFProgramma_Ciclo_Lastra();
				TFWorkFlowCase(ADR(WorkFlow[NumeroWF]),30,WorkflowCase_JMP);	// Case con FB CON interpolazione
			END_IF;
		(* Case 20 - Chiamata FB del ciclo di lavoro *)	
		20:	
			TFWorkFlowCase(ADR(WorkFlow[NumeroWF]),30,WorkflowCase_JMP);	// Case con FB CON interpolazione

			
		(* Case 30 - Chiamata FB del ciclo di lavoro *)	
		30:	
			IF CmdExe.RapidStopRequest > 0 OR
				TFPalletizerIsModuleError(Modules) OR Error.Code <> 0 THEN
				TFCiclo_Prelievo_Lastra.InterrompiCiclo := TRUE;
			ELSE
				TFCiclo_Prelievo_Lastra.InterrompiCiclo := FALSE;
			END_IF
			TFCiclo_Prelievo_Lastra.Ciclo					:= ADR(Ciclo_Prelievo_Lastra);
			TFCiclo_Prelievo_Lastra.Programma				:= ADR(TFProgramma_Ciclo_Lastra);
			TFCiclo_Prelievo_Lastra.Modules 				:= Modules;
			TFCiclo_Prelievo_Lastra.StartInterpolazioneAssi := ADR(STARTInterpolazioneASSI^);
			TFCiclo_Prelievo_Lastra.AbilitazioneAnticipoDinamicoMovimenti 	:= AbilitaAnticipoDinamico^;
			TFCiclo_Prelievo_Lastra.AbilitazioneGlobalePassMode 			:= Traiettoria^.PassModeGlobalEnable;
			TFCiclo_Prelievo_Lastra.Abilita_Ciclo_Step						:= AbilitazioCiclo_TEST_STEP;
			TFCiclo_Prelievo_Lastra.PrelievoPezzoOrizzontale				:= TRUE;
			TFCiclo_Prelievo_Lastra.NumeroTentativiPresa					:= HMI_NumeroTentativiPresa;
			
			IF CommandSTEP AND NOT CommandSTEPTRIG THEN
				TFCiclo_Prelievo_Lastra.Command_Step	:= TRUE;
				CommandSTEPTRIG := TRUE;
			ELSIF NOT CommandSTEP AND NOT CommandSTEPTRIG THEN
				TFCiclo_Prelievo_Lastra.Command_Step	:= FALSE;
				CommandSTEPTRIG := FALSE;
				CommandSTEP := FALSE;
			ELSIF  STEPCicloDONE THEN
				TFCiclo_Prelievo_Lastra.Command_Step	:= FALSE;
				CommandSTEP := FALSE;
				CommandSTEPTRIG := FALSE;
			END_IF
			
			TFCiclo_Prelievo_Lastra();
			STEPCicloDONE := TFCiclo_Prelievo_Lastra.STEPDone;
			
			IF Ciclo_Prelievo_Lastra.Stato = TERMINATO THEN
				ProductOnGripper := KPRODUCTLOADED;
				TFWorkFlowCase(ADR(WorkFlow[NumeroWF]),100,WorkflowCase_JMP);
			ELSIF Ciclo_Prelievo_Lastra.Stato = INTERROTTO THEN	
				TFWorkFlowCase(ADR(WorkFlow[NumeroWF]),999,WorkflowCase_JMP);		
			END_IF

		(* Case 100 *)
		100:WorkFlow[NumeroWF].State := StateWF_END;
			WorkFlow[NumeroWF].Enable := FALSE;
			CommandSTEP := FALSE;
			CommandSTEPTRIG := FALSE;
			AssiInterpolati := FALSE;

		(* Case 999 *)
		(* WorkFlow ERROR *)
		StateWF_ERROR:
			TFWorkFlowError(ADR(WorkFlow[NumeroWF]),ADR(WorkFlowErrorLog[NumeroWF]));
			CmdExe.PhaseStopRequest := 1;
			CmdExe.RapidStopRequest := 1;
			WorkFlow[NumeroWF].Enable := FALSE;
			CommandSTEP := FALSE;
			CommandSTEPTRIG := FALSE;
			AssiInterpolati := FALSE;
		
		ELSE						
			TFWorkFlowError(ADR(WorkFlow[NumeroWF]),ADR(WorkFlowErrorLog[NumeroWF]));
			TFError(ErrNOCMDCASE,ErrNULL,ADR(CmdExe),ADR(State),ADR(Error),ADR(ErrorLog));	
	END_CASE;
END_IF
END_ACTION

ACTION WF06_CicloDepLastraDaPP:
(*-------------------------------------------------------------------------------------------*)
(* WorkFlow 6 -  CICLO DEPOSITO LASTRA PP *)
(*-------------------------------------------------------------------------------------------*)	
NumeroWF := 6;	
IF WorkFlow[NumeroWF].Enable THEN

	IF NOT TFCommandCaseIsEnable(ADR(CmdExe)) THEN RETURN; END_IF
	CASE WorkFlow[NumeroWF].WFCase OF

		(* Case 0 *)
		0:  WorkFlow[NumeroWF].State := StateWF_RUN;
			STEPCicloDONE := FALSE;	
			TFWorkFlowCase(ADR(WorkFlow[NumeroWF]),1,WorkflowCase_INC);
	
		(* Case 1 - Chiamata del FB del ciclo di riposo per Valorizzarne i valori*)
		1:	IF CmdExe.RapidStopRequest > 0  OR
				TFPalletizerIsModuleError(Modules) THEN
				TFWorkFlowCase(ADR(WorkFlow[NumeroWF]),100,WorkflowCase_JMP);
			ELSE

				TFProgramma_Ciclo_Lastra.X_Par := ParametriProgramma_X_CicloLastra;
				TFProgramma_Ciclo_Lastra.Y_Par := ParametriProgramma_Y_CicloLastra;
				TFProgramma_Ciclo_Lastra.Z_Par := ParametriProgramma_Z_CicloLastra;
				TFProgramma_Ciclo_Lastra.J_Par := ParametriProgramma_J_CicloLastra;
				
				(*X*)
				TFProgramma_Ciclo_Lastra.Quota_StartLenta_Prelievo_Lastra_X			:= Traiettoria^.PuntoDiApproccioStartPoint.X;
				TFProgramma_Ciclo_Lastra.Quota_Prelievo_Lastra_X 					:= Traiettoria^.StartPoint.X;
				TFProgramma_Ciclo_Lastra.Quota_StartLenta_Deposito_Lastra_X	 		:= Traiettoria^.PuntoDiApproccioEndPoint.X;	
				TFProgramma_Ciclo_Lastra.Quota_Deposito_Lastra_X 					:= Traiettoria^.EndPoint.X;
				TFProgramma_Ciclo_Lastra.Quota_Fuori_Ingombro_SenzaCarico_X			:= Traiettoria^.EndPoint.X;//STESSA QUOTA DI DEPOSITO X DEPAL UNIVERSAL
				TFProgramma_Ciclo_Lastra.Quota_Fuori_Ingombro_Carico_X				:= Traiettoria^.EndPoint.X;//STESSA QUOTA DI DEPOSITO X DEPAL UNIVERSAL
				
				(*Y*)
				TFProgramma_Ciclo_Lastra.Quota_StartLenta_Prelievo_Lastra_Y         := Traiettoria^.PuntoDiApproccioStartPoint.Y;;
				TFProgramma_Ciclo_Lastra.Quota_Prelievo_Lastra_Y 					:= Traiettoria^.StartPoint.Y;
				TFProgramma_Ciclo_Lastra.Quota_Distacco_Lastra_Y					:= Traiettoria^.PuntoDiPostPosizionamentoStartPoint.Y;
				TFProgramma_Ciclo_Lastra.Quota_StartLenta_Deposito_Lastra_Y			:= Traiettoria^.PuntoDiApproccioEndPoint.Y;
				TFProgramma_Ciclo_Lastra.Quota_Deposito_Lastra_Y 					:= Traiettoria^.EndPoint.Y;
				TFProgramma_Ciclo_Lastra.Quota_Fuori_Ingombro_Y 					:= QuotaFuoriIngombro_Y_ConCARICO;//DEVE ESSERE GUALE A QUELLE DEL CORRIDOIO
				
				(*Z*)
				TFProgramma_Ciclo_Lastra.Quota_StartLenta_Prelievo_Lastra_Z 		:= MAX(Traiettoria^.PuntoDiApproccioStartPoint.Z,AxisPar_Z.MinPosition);
				TFProgramma_Ciclo_Lastra.Quota_Prelievo_Lastra_Z 					:= MAX(Traiettoria^.StartPoint.Z,AxisPar_Z.MinPosition);
				TFProgramma_Ciclo_Lastra.Quota_StartLenta_Deposito_Lastra_Z			:= Traiettoria^.PuntoDiApproccioEndPoint.Z;
				TFProgramma_Ciclo_Lastra.Quota_Deposito_Lastra_Z					:= Traiettoria^.EndPoint.Z;
				TFProgramma_Ciclo_Lastra.Quota_Fuori_Ingombro_ConCarico_Z			:= QuotaFuoriIngombro_Z_ConPEZZO;
				TFProgramma_Ciclo_Lastra.Quota_Fuori_Ingombro_SenzaCarico_Z			:= QuotaFuoriIngombro_Z_AVUOTO;
				TFProgramma_Ciclo_Lastra.Quota_Distacco_Lastra_Z					:= Traiettoria^.PuntoDiPostPosizionamentoStartPoint.Z;
				TFProgramma_Ciclo_Lastra.Quota_PostScarico							:= Z_Riposo;	
			
				(*J*)
				TFProgramma_Ciclo_Lastra.Quota_Rotazione_Prelievo_Lastra 			:= Traiettoria^.StartPoint.J;
				TFProgramma_Ciclo_Lastra.Quota_Rotazione_Deposito_Lastra 			:= Traiettoria^.EndPoint.J;
				TFProgramma_Ciclo_Lastra.Quota_Rotazione_StartTasteggio_Lastra		:= Traiettoria^.PuntoDiApproccioStartPoint.J;
				TFProgramma_Ciclo_Lastra.Quota_Fuori_Ingombro_J						:= QuotaFuoriIngombro_J_ConCARICO;
				TFProgramma_Ciclo_Lastra.Quota_Rotazione_Sfogliatura 				:= Traiettoria^.StartPoint.J + HMI_GradiSfogliaturaJ;

				TFProgramma_Ciclo_Lastra();
				TFWorkFlowCase(ADR(WorkFlow[NumeroWF]),30,WorkflowCase_JMP);	// Case con FB CON interpolazione
			END_IF;
		(* Case 20 - Chiamata FB del ciclo di lavoro *)	
		20:	
			TFWorkFlowCase(ADR(WorkFlow[NumeroWF]),30,WorkflowCase_JMP);	// Case con FB CON interpolazione

			
		(* Case 30 - Chiamata FB del ciclo di lavoro *)	
		30:	
			IF CmdExe.RapidStopRequest > 0 OR
				TFPalletizerIsModuleError(Modules) THEN
				TFCiclo_Deposito_Lastra.InterrompiCiclo := TRUE;
			ELSE
				TFCiclo_Deposito_Lastra.InterrompiCiclo := FALSE;
			END_IF
			TFCiclo_Deposito_Lastra.Ciclo					:= ADR(Ciclo_Deposito_Lastra);
			TFCiclo_Deposito_Lastra.Programma				:= ADR(TFProgramma_Ciclo_Lastra);
			TFCiclo_Deposito_Lastra.ModuleAX_X 				:= ADR(Modules^.AX_X);
			TFCiclo_Deposito_Lastra.ModuleAX_Y 				:= ADR(Modules^.AX_Y);
			TFCiclo_Deposito_Lastra.ModuleAX_Z 				:= ADR(Modules^.AX_Z);
			TFCiclo_Deposito_Lastra.ModuleAX_J 				:= ADR(Modules^.AX_J);
			TFCiclo_Deposito_Lastra.ModulePinza 			:= ADR(Modules^.Pinza);
			TFCiclo_Deposito_Lastra.StartInterpolazioneAssi := ADR(STARTInterpolazioneASSI^);
			TFCiclo_Deposito_Lastra.AbilitazioneAnticipoDinamicoMovimenti 	:= AbilitaAnticipoDinamico^;
			TFCiclo_Deposito_Lastra.AbilitazioneGlobalePassMode 			:= Traiettoria^.PassModeGlobalEnable;
			TFCiclo_Deposito_Lastra.Abilita_Ciclo_Step						:= AbilitazioCiclo_TEST_STEP;
			
			IF CommandSTEP AND NOT CommandSTEPTRIG THEN
				TFCiclo_Deposito_Lastra.Command_Step	:= TRUE;
				CommandSTEPTRIG := TRUE;
			ELSIF NOT CommandSTEP AND NOT CommandSTEPTRIG THEN
				TFCiclo_Deposito_Lastra.Command_Step	:= FALSE;
				CommandSTEPTRIG := FALSE;
				CommandSTEP := FALSE;
			ELSIF  STEPCicloDONE THEN
				TFCiclo_Deposito_Lastra.Command_Step	:= FALSE;
				CommandSTEP := FALSE;
				CommandSTEPTRIG := FALSE;
			END_IF
			
			TFCiclo_Deposito_Lastra();
			STEPCicloDONE := TFCiclo_Deposito_Lastra.STEPDone;
			
			IF Ciclo_Deposito_Lastra.Stato = TERMINATO THEN
				ProductOnGripper := KNOPRODUCT;
				TFWorkFlowCase(ADR(WorkFlow[NumeroWF]),100,WorkflowCase_JMP);
			ELSIF Ciclo_Deposito_Lastra.Stato = INTERROTTO THEN	
				TFWorkFlowCase(ADR(WorkFlow[NumeroWF]),999,WorkflowCase_JMP);		
			END_IF

		(* Case 100 *)
		100:WorkFlow[NumeroWF].State := StateWF_END;
			WorkFlow[NumeroWF].Enable := FALSE;
			CommandSTEP := FALSE;
			CommandSTEPTRIG := FALSE;
			AssiInterpolati := FALSE;

		(* Case 999 *)
		(* WorkFlow ERROR *)
		StateWF_ERROR:
			TFWorkFlowError(ADR(WorkFlow[NumeroWF]),ADR(WorkFlowErrorLog[NumeroWF]));
			CmdExe.PhaseStopRequest := 1;
			CmdExe.RapidStopRequest := 1;
			WorkFlow[NumeroWF].Enable := FALSE;
			CommandSTEP := FALSE;
			CommandSTEPTRIG := FALSE;
			AssiInterpolati := FALSE;
		
		ELSE						
			TFWorkFlowError(ADR(WorkFlow[NumeroWF]),ADR(WorkFlowErrorLog[NumeroWF]));
			TFError(ErrNOCMDCASE,ErrNULL,ADR(CmdExe),ADR(State),ADR(Error),ADR(ErrorLog));	
	END_CASE;
END_IF
END_ACTION

ACTION WF07_CicloPrelLastraDaWA:
(*-------------------------------------------------------------------------------------------*)
(* WorkFlow 7 -  CICLO PRELIEVO LASTRA DA WA *)
(*-------------------------------------------------------------------------------------------*)	
NumeroWF := 7;	
IF WorkFlow[NumeroWF].Enable THEN

	IF NOT TFCommandCaseIsEnable(ADR(CmdExe)) THEN RETURN; END_IF
	CASE WorkFlow[NumeroWF].WFCase OF

		(* Case 0 *)
		0:  WorkFlow[NumeroWF].State := StateWF_RUN;
			STEPCicloDONE := FALSE;	
			OUT.StartTilter := TRUE;
			TFWorkFlowCase(ADR(WorkFlow[NumeroWF]),1,WorkflowCase_INC);
	
		(* Case 1 - Chiamata del FB del ciclo di riposo per Valorizzarne i valori*)
		1:	IF CmdExe.RapidStopRequest > 0  OR
				TFPalletizerIsModuleError(Modules) THEN
				TFWorkFlowCase(ADR(WorkFlow[NumeroWF]),100,WorkflowCase_JMP);
			ELSE

				TFProgramma_Ciclo_Lastra.X_Par := ParametriProgramma_X_CicloLastra;
				TFProgramma_Ciclo_Lastra.Y_Par := ParametriProgramma_Y_CicloLastra;
				TFProgramma_Ciclo_Lastra.Z_Par := ParametriProgramma_Z_CicloLastra;
				TFProgramma_Ciclo_Lastra.J_Par := ParametriProgramma_J_CicloLastra;
				
				(*X*)
				TFProgramma_Ciclo_Lastra.Quota_StartLenta_Prelievo_Lastra_X			:= Traiettoria^.PuntoDiApproccioStartPoint.X;
				TFProgramma_Ciclo_Lastra.Quota_Prelievo_Lastra_X 					:= Traiettoria^.StartPoint.X;
				TFProgramma_Ciclo_Lastra.Quota_StartLenta_Deposito_Lastra_X	 		:= Traiettoria^.PuntoDiApproccioEndPoint.X;	
				TFProgramma_Ciclo_Lastra.Quota_Deposito_Lastra_X 					:= Traiettoria^.EndPoint.X;
				TFProgramma_Ciclo_Lastra.Quota_Fuori_Ingombro_SenzaCarico_X			:= Traiettoria^.StartPoint.X;
				TFProgramma_Ciclo_Lastra.Quota_Fuori_Ingombro_Carico_X				:= Traiettoria^.StartPoint.X;
				//*****************************************************************
				CoordenadaPosGiroPieza_X := WorkArea^[NuPosGuiroPiking].X ;
				TFProgramma_Ciclo_Lastra.Quota_PosGiroPiezaTraCavalleteX			:= CoordenadaPosGiroPieza_X ;
				//*****************************************************************
				(*Y*)
				TFProgramma_Ciclo_Lastra.Quota_StartLenta_Prelievo_Lastra_Y         := Traiettoria^.PuntoDiApproccioStartPoint.Y;;
				TFProgramma_Ciclo_Lastra.Quota_Prelievo_Lastra_Y 					:= Traiettoria^.StartPoint.Y;
				TFProgramma_Ciclo_Lastra.Quota_Distacco_Lastra_Y					:= Traiettoria^.PuntoDiPostPosizionamentoStartPoint.Y;
				TFProgramma_Ciclo_Lastra.Quota_StartLenta_Deposito_Lastra_Y			:= Traiettoria^.PuntoDiApproccioEndPoint.Y;
				TFProgramma_Ciclo_Lastra.Quota_Deposito_Lastra_Y 					:= Traiettoria^.EndPoint.Y;
				TFProgramma_Ciclo_Lastra.Quota_Fuori_Ingombro_Y 					:= QuotaFuoriIngombro_Y_AVUOTO;
				TFProgramma_Ciclo_Lastra.Quota_PasilloCavallete0GradosY             := CoordenadaPasillo0_Y ;
				TFProgramma_Ciclo_Lastra.Quota_PasilloCavallete1800GradosY          := CoordenadaPasillo180_Y ;
				
				(*Z*)
				TFProgramma_Ciclo_Lastra.Quota_StartLenta_Prelievo_Lastra_Z 		:= MAX(Traiettoria^.PuntoDiApproccioStartPoint.Z,AxisPar_Z.MinPosition+1);
				TFProgramma_Ciclo_Lastra.Quota_Prelievo_Lastra_Z 					:= MAX(Traiettoria^.StartPoint.Z,AxisPar_Z.MinPosition+1);
				TFProgramma_Ciclo_Lastra.Quota_StartLenta_Deposito_Lastra_Z			:= Traiettoria^.PuntoDiApproccioEndPoint.Z;
				TFProgramma_Ciclo_Lastra.Quota_Deposito_Lastra_Z					:= MAX(Traiettoria^.EndPoint.Z,AxisPar_Z.MinPosition+1);
				TFProgramma_Ciclo_Lastra.Quota_Fuori_Ingombro_ConCarico_Z			:= QuotaFuoriIngombro_Z_ConPEZZO;
				TFProgramma_Ciclo_Lastra.Quota_Fuori_Ingombro_SenzaCarico_Z			:= QuotaFuoriIngombro_Z_AVUOTO;
				TFProgramma_Ciclo_Lastra.Quota_Distacco_Lastra_Z					:= Traiettoria^.PuntoDiPostPosizionamentoStartPoint.Z;
				TFProgramma_Ciclo_Lastra.Quota_PostScarico							:= Z_Riposo;	
			
				(*J*)
				TFProgramma_Ciclo_Lastra.Quota_Rotazione_Prelievo_Lastra 			:= Traiettoria^.StartPoint.J;
				TFProgramma_Ciclo_Lastra.Quota_Rotazione_Deposito_Lastra 			:= Traiettoria^.EndPoint.J;
				TFProgramma_Ciclo_Lastra.Quota_Rotazione_StartTasteggio_Lastra		:= Traiettoria^.StartPoint.J;
				TFProgramma_Ciclo_Lastra.Quota_Fuori_Ingombro_J						:= QuotaFuoriIngombro_J_AVUOTO;
				TFProgramma_Ciclo_Lastra.Quota_Rotazione_Sfogliatura 				:= Traiettoria^.StartPoint.J + HMI_GradiSfogliaturaJ;
				TFProgramma_Ciclo_Lastra.Quota_Fuori_Ingombro_AttualeJ 				:= QuotaFuoriIngombro_J_AVUOTO;

				TFProgramma_Ciclo_Lastra();
				CommandSTEP := FALSE;
				TFWorkFlowCase(ADR(WorkFlow[NumeroWF]),30,WorkflowCase_JMP);	// Case con FB CON interpolazione
			END_IF;
		(* Case 20 - Chiamata FB del ciclo di lavoro *)	
		20:	
			TFWorkFlowCase(ADR(WorkFlow[NumeroWF]),30,WorkflowCase_JMP);	// Case con FB CON interpolazione

			
		(* Case 30 - Chiamata FB del ciclo di lavoro *)	
		30:	
			IF CmdExe.RapidStopRequest > 0 OR
				TFPalletizerIsModuleError(Modules) OR Error.Code <> 0 THEN
				TFCiclo_Prelievo_Lastra.InterrompiCiclo := TRUE;
			ELSE
				TFCiclo_Prelievo_Lastra.InterrompiCiclo := FALSE;
			END_IF

			TFCiclo_Prelievo_Lastra.Ciclo									:= ADR(Ciclo_Prelievo_Lastra);
			TFCiclo_Prelievo_Lastra.Programma								:= ADR(TFProgramma_Ciclo_Lastra);
			TFCiclo_Prelievo_Lastra.Modules	 								:= Modules;
			TFCiclo_Prelievo_Lastra.StartInterpolazioneAssi 				:= ADR(STARTInterpolazioneASSI^);
			TFCiclo_Prelievo_Lastra.AbilitazioneAnticipoDinamicoMovimenti 	:= AbilitaAnticipoDinamico^;
			TFCiclo_Prelievo_Lastra.AbilitazioneGlobalePassMode 			:= Traiettoria^.PassModeGlobalEnable;
			TFCiclo_Prelievo_Lastra.Abilita_Ciclo_Step						:= AbilitazioCiclo_TEST_STEP;
			TFCiclo_Prelievo_Lastra.PrelievoPezzoOrizzontale				:= Mission^.JPick = 90;
			TFCiclo_Prelievo_Lastra.NumeroTentativiPresa					:= HMI_NumeroTentativiPresa;
			TFCiclo_Prelievo_Lastra.Mission									:= Mission;
			//TFCiclo_Prelievo_Lastra.Quota_Rotazione_StartTasteggio_Lastra   := Quota_Rotazione_StartTasteggio_Lastra ;
			IF CommandSTEP AND NOT CommandSTEPTRIG THEN
				TFCiclo_Prelievo_Lastra.Command_Step	:= TRUE;
				CommandSTEPTRIG := TRUE;
			ELSIF NOT CommandSTEP AND NOT CommandSTEPTRIG THEN
				TFCiclo_Prelievo_Lastra.Command_Step	:= FALSE;
				CommandSTEPTRIG := FALSE;
				CommandSTEP := FALSE;
			ELSIF  STEPCicloDONE THEN
				TFCiclo_Prelievo_Lastra.Command_Step	:= FALSE;
				CommandSTEP := FALSE;
				CommandSTEPTRIG := FALSE;
			END_IF
			
			TFCiclo_Prelievo_Lastra();
			STEPCicloDONE := TFCiclo_Prelievo_Lastra.STEPDone;
			
			IF TFCiclo_Prelievo_Lastra.Ciclo^.Stato = TERMINATO THEN
				ProductOnGripper := KPRODUCTLOADED;
				TFWorkFlowCase(ADR(WorkFlow[NumeroWF]),100,WorkflowCase_JMP);
			ELSIF TFCiclo_Prelievo_Lastra.Errore > 0 THEN
				TFError(TFCiclo_Prelievo_Lastra.Errore,ErrNULL,ADR(CmdExe),ADR(State),ADR(Error),ADR(ErrorLog));	
				TFWorkFlowCase(ADR(WorkFlow[NumeroWF]),999,WorkflowCase_JMP);	 
			ELSIF TFCiclo_Prelievo_Lastra.Ciclo^.Stato = INTERROTTO THEN	
				TFWorkFlowCase(ADR(WorkFlow[NumeroWF]),999,WorkflowCase_JMP);		
			END_IF

		(* Case 100 *)
		100:WorkFlow[NumeroWF].State := StateWF_END;
			WorkFlow[NumeroWF].Enable := FALSE;
			CommandSTEP := FALSE;
			CommandSTEPTRIG := FALSE;
			AssiInterpolati := FALSE;

		(* Case 999 *)
		(* WorkFlow ERROR *)
		StateWF_ERROR:
			TFWorkFlowError(ADR(WorkFlow[NumeroWF]),ADR(WorkFlowErrorLog[NumeroWF]));
			CmdExe.PhaseStopRequest := 1;
			CmdExe.RapidStopRequest := 1;
			WorkFlow[NumeroWF].Enable := FALSE;
			CommandSTEP := FALSE;
			CommandSTEPTRIG := FALSE;
			AssiInterpolati := FALSE;
		
		ELSE						
			TFWorkFlowError(ADR(WorkFlow[NumeroWF]),ADR(WorkFlowErrorLog[NumeroWF]));
			TFError(ErrNOCMDCASE,ErrNULL,ADR(CmdExe),ADR(State),ADR(Error),ADR(ErrorLog));	
	END_CASE;
END_IF
END_ACTION

ACTION WF08_CicloDepLastraSuPareggiatore:
(*-------------------------------------------------------------------------------------------*)
(* WorkFlow 8 -  CICLO DEPOSITO LASTRA SU PAREGGIATORE *)
(*-------------------------------------------------------------------------------------------*)		
NumeroWF := 8;
IF WorkFlow[NumeroWF].Enable THEN

	IF NOT TFCommandCaseIsEnable(ADR(CmdExe)) THEN RETURN; END_IF
	CASE WorkFlow[NumeroWF].WFCase OF

		(* Case 0 *)
		0:  WorkFlow[NumeroWF].State := StateWF_RUN;
			STEPCicloDONE := FALSE;
			OUT.StartTilter := TRUE;
			PaccoPresoXDataLogger := FALSE;
			IF NOT AttivaTimerContaPacchi1Minuto THEN
				AttivaTimerContaPacchi1Minuto := TRUE;
				AttivaTimerContaPacchi5Minuti := TRUE;
				Pacchi1Minuto := Pacchi1Minuto +1;
			ELSIF AttivaTimerContaPacchi1Minuto THEN
				AttivaTimerContaPacchi1Minuto := TRUE;
				Pacchi1Minuto := Pacchi1Minuto +1;
			END_IF	
			
			TFWorkFlowCase(ADR(WorkFlow[NumeroWF]),1,WorkflowCase_INC);
	
		(* Case 1 - Chiamata del FB del ciclo di riposo per Valorizzarne i valori*)
		1:	IF CmdExe.RapidStopRequest > 0 OR
				TFPalletizerIsModuleError(Modules) THEN
				TFWorkFlowCase(ADR(WorkFlow[NumeroWF]),100,WorkflowCase_JMP);
			ELSE
				TFProgramma_Ciclo_Lastra.X_Par := ParametriProgramma_X_CicloLastra;
				TFProgramma_Ciclo_Lastra.Y_Par := ParametriProgramma_Y_CicloLastra;
				TFProgramma_Ciclo_Lastra.Z_Par := ParametriProgramma_Z_CicloLastra;
				TFProgramma_Ciclo_Lastra.J_Par := ParametriProgramma_J_CicloLastra;
				
				(*X*)
				TFProgramma_Ciclo_Lastra.Quota_Prelievo_Lastra_X 					:= Traiettoria^.StartPoint.X;
				TFProgramma_Ciclo_Lastra.Quota_StartLenta_Deposito_Lastra_X	 		:= Traiettoria^.PuntoDiApproccioEndPoint.X;	
				TFProgramma_Ciclo_Lastra.Quota_Deposito_Lastra_X 					:= Traiettoria^.EndPoint.X;
				
				(*Y*)
				TFProgramma_Ciclo_Lastra.Quota_Prelievo_Lastra_Y 					:= Traiettoria^.StartPoint.Y;
				TFProgramma_Ciclo_Lastra.Quota_StartLenta_Deposito_Lastra_Y			:= Traiettoria^.PuntoDiApproccioEndPoint.Y;
				TFProgramma_Ciclo_Lastra.Quota_Deposito_Lastra_Y 					:= Traiettoria^.EndPoint.Y;
				TFProgramma_Ciclo_Lastra.Quota_Fuori_Ingombro_Y 					:= QuotaFuoriIngombroColonne_Y;//(WorkSpace^.Y - IngombroSuperficialePinzaMAX_Global/2);
				
				(*Z*)
				TFProgramma_Ciclo_Lastra.Quota_StartLenta_Prelievo_Lastra_Z 			:= Traiettoria^.PuntoDiApproccioStartPoint.Z;
				TFProgramma_Ciclo_Lastra.Quota_Prelievo_Lastra_Z 					:= Traiettoria^.StartPoint.Z;
				TFProgramma_Ciclo_Lastra.DisabilitaDepositoConTasteggio				:= (NOT AbilitaDepositoPaccoOrrizzonataleConTasteggio^ OR
																						SimulazioneSenzaPalletFalde);
				
